(* PLC project TemplatePLC210_03, CODESYS CODESYS V3.5 SP14 Patch 3 *)
(* stored: creationDateTime 2022-10-11T10:43:14.2578546, version 3.5.14.30, modificationDateTime 2022-10-11T10:23:43.7157386, organization Production association OWEN *)

TYPE CTRL8 : STRUCT
  ID : BYTE := 108;
  SIZE : BYTE;
  BIT0 : BIT;
  BIT1 : BIT;
  BIT2 : BIT;
  BIT3 : BIT;
  BIT4 : BIT;
  BIT5 : BIT;
  BIT6 : BIT;
  BIT7 : BIT;
  BIT8 : BIT;
  BIT9 : BIT;
  BIT10 : BIT;
  BIT11 : BIT;
  BIT12 : BIT;
  BIT13 : BIT;
  BIT14 : BIT;
  BIT15 : BIT;
END_STRUCT;
END_TYPE

TYPE bCTRL8 : STRUCT
  CTRL : ARRAY[0..3] OF BYTE;
END_STRUCT;
END_TYPE

TYPE CTRL16 : STRUCT
  ID : WORD := 116;
  SIZE : WORD;
  BIT0 : BIT;
  BIT1 : BIT;
  BIT2 : BIT;
  BIT3 : BIT;
  BIT4 : BIT;
  BIT5 : BIT;
  BIT6 : BIT;
  BIT7 : BIT;
  BIT8 : BIT;
  BIT9 : BIT;
  BIT10 : BIT;
  BIT11 : BIT;
  BIT12 : BIT;
  BIT13 : BIT;
  BIT14 : BIT;
  BIT15 : BIT;
  BIT16 : BIT;
  BIT17 : BIT;
  BIT18 : BIT;
  BIT19 : BIT;
  BIT20 : BIT;
  BIT21 : BIT;
  BIT22 : BIT;
  BIT23 : BIT;
  BIT24 : BIT;
  BIT25 : BIT;
  BIT26 : BIT;
  BIT27 : BIT;
  BIT28 : BIT;
  BIT29 : BIT;
  BIT30 : BIT;
  BIT31 : BIT;
END_STRUCT;
END_TYPE

TYPE wCTRL16 : STRUCT
  CTRL : ARRAY[0..3] OF WORD;
END_STRUCT;
END_TYPE

TYPE CTRL32 : STRUCT
  ID : DWORD := 132;
  SIZE : DWORD;
  BIT0 : BIT;
  BIT1 : BIT;
  BIT2 : BIT;
  BIT3 : BIT;
  BIT4 : BIT;
  BIT5 : BIT;
  BIT6 : BIT;
  BIT7 : BIT;
  BIT8 : BIT;
  BIT9 : BIT;
  BIT10 : BIT;
  BIT11 : BIT;
  BIT12 : BIT;
  BIT13 : BIT;
  BIT14 : BIT;
  BIT15 : BIT;
  BIT16 : BIT;
  BIT17 : BIT;
  BIT18 : BIT;
  BIT19 : BIT;
  BIT20 : BIT;
  BIT21 : BIT;
  BIT22 : BIT;
  BIT23 : BIT;
  BIT24 : BIT;
  BIT25 : BIT;
  BIT26 : BIT;
  BIT27 : BIT;
  BIT28 : BIT;
  BIT29 : BIT;
  BIT30 : BIT;
  BIT31 : BIT;
  BIT32 : BIT;
  BIT33 : BIT;
  BIT34 : BIT;
  BIT35 : BIT;
  BIT36 : BIT;
  BIT37 : BIT;
  BIT38 : BIT;
  BIT39 : BIT;
  BIT40 : BIT;
  BIT41 : BIT;
  BIT42 : BIT;
  BIT43 : BIT;
  BIT44 : BIT;
  BIT45 : BIT;
  BIT46 : BIT;
  BIT47 : BIT;
  BIT48 : BIT;
  BIT49 : BIT;
  BIT50 : BIT;
  BIT51 : BIT;
  BIT52 : BIT;
  BIT53 : BIT;
  BIT54 : BIT;
  BIT55 : BIT;
  BIT56 : BIT;
  BIT57 : BIT;
  BIT58 : BIT;
  BIT59 : BIT;
  BIT60 : BIT;
  BIT61 : BIT;
  BIT62 : BIT;
  BIT63 : BIT;
END_STRUCT;
END_TYPE

TYPE dwCTRL32 : STRUCT
  CTRL : ARRAY[0..3] OF DWORD;
END_STRUCT;
END_TYPE

TYPE uCTRL8 : UNION
  _CTRL8 : CTRL8;
  _wCTRL8 : bCTRL8;
END_UNION;
END_TYPE

TYPE uCTRL16 : UNION
  _CTRL16 : CTRL16;
  _wCTRL16 : wCTRL16;
END_UNION;
END_TYPE

TYPE uCTRL32 : UNION
  _CTRL32 : CTRL32;
  _dwCTRL32 : dwCTRL32;
END_UNION;
END_TYPE

FUNCTION AND16 : BOOL
  VAR_INPUT
    IN_ADR1 : POINTER TO WORD;
    IN_ADR2 : POINTER TO WORD;
    OUT_ADR3 : POINTER TO WORD;
  END_VAR
  VAR
    SIZE : WORD;
    pwADR1 : POINTER TO WORD;
    pwADR2 : POINTER TO WORD;
    pwADR3 : POINTER TO WORD;
    COUNT : WORD;
  END_VAR
  VAR CONSTANT
    STEP : WORD := 2;
  END_VAR

            	pwADR1	:=	IN_ADR1+STEP;
	SIZE	:=	pwADR1^;
IF IN_ADR1^ = IN_ADR2^ AND IN_ADR1^ = OUT_ADR3^ AND SIZE MOD STEP = 0 THEN
	FOR COUNT:=2*STEP TO SIZE-STEP BY STEP DO
		pwADR1	:=	IN_ADR1+COUNT;
		pwADR2	:=	IN_ADR2+COUNT;
		pwADR3	:=	OUT_ADR3+COUNT;
		pwADR3^ := pwADR1^ AND pwADR2^;
	END_FOR
ELSE
	AND16	:=	TRUE;
END_IF

          
END_FUNCTION

FUNCTION AND32 : BOOL
  VAR_INPUT
    IN_ADR1 : POINTER TO DWORD;
    IN_ADR2 : POINTER TO DWORD;
    OUT_ADR3 : POINTER TO DWORD;
  END_VAR
  VAR
    SIZE : DWORD;
    pdwADR1 : POINTER TO DWORD;
    pdwADR2 : POINTER TO DWORD;
    pdwADR3 : POINTER TO DWORD;
    COUNT : DWORD;
  END_VAR
  VAR CONSTANT
    STEP : DWORD := 4;
  END_VAR

            	pdwADR1	:=	IN_ADR1+STEP;
	SIZE	:=	pdwADR1^;
IF IN_ADR1^ = IN_ADR2^ AND IN_ADR1^ = OUT_ADR3^ AND SIZE MOD STEP = 0 THEN
	FOR COUNT:=2*STEP TO SIZE-STEP BY STEP DO
		pdwADR1	:=	IN_ADR1+COUNT;
		pdwADR2	:=	IN_ADR2+COUNT;
		pdwADR3	:=	OUT_ADR3+COUNT;
		pdwADR3^ := pdwADR1^ AND pdwADR2^;
	END_FOR
ELSE
	AND32	:=	TRUE;
END_IF
          
END_FUNCTION

FUNCTION AND8 : BOOL
  VAR_INPUT
    IN_ADR1 : POINTER TO BYTE;
    IN_ADR2 : POINTER TO BYTE;
    OUT_ADR3 : POINTER TO BYTE;
  END_VAR
  VAR
    SIZE : BYTE;
    pbADR1 : POINTER TO BYTE;
    pbADR2 : POINTER TO BYTE;
    pbADR3 : POINTER TO BYTE;
    COUNT : BYTE;
  END_VAR

            IF IN_ADR1^ = IN_ADR2^ AND IN_ADR1^ = OUT_ADR3^ THEN
	pbADR1	:=	IN_ADR1+1;
	SIZE	:=	pbADR1^;
	FOR COUNT:=2 TO SIZE-1 DO
		pbADR1	:=	IN_ADR1+COUNT;
		pbADR2	:=	IN_ADR2+COUNT;
		pbADR3	:=	OUT_ADR3+COUNT;
		pbADR3^ := pbADR1^ AND pbADR2^;
	END_FOR
ELSE
	AND8	:=	TRUE;
END_IF

          
END_FUNCTION

FUNCTION NAND8 : BOOL
  VAR_INPUT
    IN_ADR1 : POINTER TO BYTE;
    IN_ADR2 : POINTER TO BYTE;
    OUT_ADR3 : POINTER TO BYTE;
  END_VAR
  VAR
    SIZE : BYTE;
    pbADR1 : POINTER TO BYTE;
    pbADR2 : POINTER TO BYTE;
    pbADR3 : POINTER TO BYTE;
    COUNT : BYTE;
  END_VAR

            IF IN_ADR1^ = IN_ADR2^ AND IN_ADR1^ = OUT_ADR3^ THEN
	pbADR1	:=	IN_ADR1+1;
	SIZE	:=	pbADR1^;
	FOR COUNT:=2 TO SIZE-1 DO
		pbADR1	:=	IN_ADR1+COUNT;
		pbADR2	:=	IN_ADR2+COUNT;
		pbADR3	:=	OUT_ADR3+COUNT;
		pbADR3^ := NOT(pbADR1^ AND pbADR2^);
	END_FOR
ELSE
	NAND8	:=	TRUE;
END_IF

          
END_FUNCTION

FUNCTION NAND16 : BOOL
  VAR_INPUT
    IN_ADR1 : POINTER TO WORD;
    IN_ADR2 : POINTER TO WORD;
    OUT_ADR3 : POINTER TO WORD;
  END_VAR
  VAR
    SIZE : WORD;
    pwADR1 : POINTER TO WORD;
    pwADR2 : POINTER TO WORD;
    pwADR3 : POINTER TO WORD;
    COUNT : WORD;
  END_VAR
  VAR CONSTANT
    STEP : WORD := 2;
  END_VAR

            	pwADR1	:=	IN_ADR1+STEP;
	SIZE	:=	pwADR1^;
IF IN_ADR1^ = IN_ADR2^ AND IN_ADR1^ = OUT_ADR3^ AND SIZE MOD STEP = 0 THEN
	FOR COUNT:=2*STEP TO SIZE-STEP BY STEP DO
		pwADR1	:=	IN_ADR1+COUNT;
		pwADR2	:=	IN_ADR2+COUNT;
		pwADR3	:=	OUT_ADR3+COUNT;
		pwADR3^ := NOT(pwADR1^ AND pwADR2^);
	END_FOR
ELSE
	NAND16	:=	TRUE;
END_IF

          
END_FUNCTION

FUNCTION NAND32 : BOOL
  VAR_INPUT
    IN_ADR1 : POINTER TO DWORD;
    IN_ADR2 : POINTER TO DWORD;
    OUT_ADR3 : POINTER TO DWORD;
  END_VAR
  VAR
    SIZE : DWORD;
    pdwADR1 : POINTER TO DWORD;
    pdwADR2 : POINTER TO DWORD;
    pdwADR3 : POINTER TO DWORD;
    COUNT : DWORD;
  END_VAR
  VAR CONSTANT
    STEP : DWORD := 4;
  END_VAR

            	pdwADR1	:=	IN_ADR1+STEP;
	SIZE	:=	pdwADR1^;
IF IN_ADR1^ = IN_ADR2^ AND IN_ADR1^ = OUT_ADR3^ AND SIZE MOD STEP = 0 THEN
	FOR COUNT:=2*STEP TO SIZE-STEP BY STEP DO
		pdwADR1	:=	IN_ADR1+COUNT;
		pdwADR2	:=	IN_ADR2+COUNT;
		pdwADR3	:=	OUT_ADR3+COUNT;
		pdwADR3^ := NOT(pdwADR1^ AND pdwADR2^);
	END_FOR
ELSE
	NAND32	:=	TRUE;
END_IF

          
END_FUNCTION

FUNCTION OR8 : BOOL
  VAR_INPUT
    IN_ADR1 : POINTER TO BYTE;
    IN_ADR2 : POINTER TO BYTE;
    OUT_ADR3 : POINTER TO BYTE;
  END_VAR
  VAR
    SIZE : BYTE;
    pbADR1 : POINTER TO BYTE;
    pbADR2 : POINTER TO BYTE;
    pbADR3 : POINTER TO BYTE;
    COUNT : BYTE;
  END_VAR

            IF IN_ADR1^ = IN_ADR2^ AND IN_ADR1^ = OUT_ADR3^ THEN
	pbADR1	:=	IN_ADR1+1;
	SIZE	:=	pbADR1^;
	FOR COUNT:=2 TO SIZE-1 DO
		pbADR1	:=	IN_ADR1+COUNT;
		pbADR2	:=	IN_ADR2+COUNT;
		pbADR3	:=	OUT_ADR3+COUNT;
		pbADR3^ := pbADR1^ OR pbADR2^;
	END_FOR
ELSE
	OR8	:=	TRUE;
END_IF

          
END_FUNCTION

FUNCTION OR16 : BOOL
  VAR_INPUT
    IN_ADR1 : POINTER TO WORD;
    IN_ADR2 : POINTER TO WORD;
    OUT_ADR3 : POINTER TO WORD;
  END_VAR
  VAR
    SIZE : WORD;
    pwADR1 : POINTER TO WORD;
    pwADR2 : POINTER TO WORD;
    pwADR3 : POINTER TO WORD;
    COUNT : WORD;
  END_VAR
  VAR CONSTANT
    STEP : WORD := 2;
  END_VAR

            	pwADR1	:=	IN_ADR1+STEP;
	SIZE	:=	pwADR1^;
IF IN_ADR1^ = IN_ADR2^ AND IN_ADR1^ = OUT_ADR3^ AND SIZE MOD STEP = 0 THEN
	FOR COUNT:=2*STEP TO SIZE-STEP BY STEP DO
		pwADR1	:=	IN_ADR1+COUNT;
		pwADR2	:=	IN_ADR2+COUNT;
		pwADR3	:=	OUT_ADR3+COUNT;
		pwADR3^ := pwADR1^ OR pwADR2^;
	END_FOR
ELSE
	OR16	:=	TRUE;
END_IF

          
END_FUNCTION

FUNCTION OR32 : BOOL
  VAR_INPUT
    IN_ADR1 : POINTER TO DWORD;
    IN_ADR2 : POINTER TO DWORD;
    OUT_ADR3 : POINTER TO DWORD;
  END_VAR
  VAR
    SIZE : DWORD;
    pdwADR1 : POINTER TO DWORD;
    pdwADR2 : POINTER TO DWORD;
    pdwADR3 : POINTER TO DWORD;
    COUNT : DWORD;
  END_VAR
  VAR CONSTANT
    STEP : DWORD := 4;
  END_VAR

            	pdwADR1	:=	IN_ADR1+STEP;
	SIZE	:=	pdwADR1^;
IF IN_ADR1^ = IN_ADR2^ AND IN_ADR1^ = OUT_ADR3^ AND SIZE MOD STEP = 0 THEN
	FOR COUNT:=2*STEP TO SIZE-STEP BY STEP DO
		pdwADR1	:=	IN_ADR1+COUNT;
		pdwADR2	:=	IN_ADR2+COUNT;
		pdwADR3	:=	OUT_ADR3+COUNT;
		pdwADR3^ := pdwADR1^ OR pdwADR2^;
	END_FOR
ELSE
	OR32	:=	TRUE;
END_IF

          
END_FUNCTION

FUNCTION NOR8 : BOOL
  VAR_INPUT
    IN_ADR1 : POINTER TO BYTE;
    IN_ADR2 : POINTER TO BYTE;
    OUT_ADR3 : POINTER TO BYTE;
  END_VAR
  VAR
    SIZE : BYTE;
    pbADR1 : POINTER TO BYTE;
    pbADR2 : POINTER TO BYTE;
    pbADR3 : POINTER TO BYTE;
    COUNT : BYTE;
  END_VAR

            IF IN_ADR1^ = IN_ADR2^ AND IN_ADR1^ = OUT_ADR3^ THEN
	pbADR1	:=	IN_ADR1+1;
	SIZE	:=	pbADR1^;
	FOR COUNT:=2 TO SIZE-1 DO
		pbADR1	:=	IN_ADR1+COUNT;
		pbADR2	:=	IN_ADR2+COUNT;
		pbADR3	:=	OUT_ADR3+COUNT;
		pbADR3^ := NOT(pbADR1^ OR pbADR2^);
	END_FOR
ELSE
	NOR8	:=	TRUE;
END_IF

          
END_FUNCTION

FUNCTION NOR16 : BOOL
  VAR_INPUT
    IN_ADR1 : POINTER TO WORD;
    IN_ADR2 : POINTER TO WORD;
    OUT_ADR3 : POINTER TO WORD;
  END_VAR
  VAR
    SIZE : WORD;
    pwADR1 : POINTER TO WORD;
    pwADR2 : POINTER TO WORD;
    pwADR3 : POINTER TO WORD;
    COUNT : WORD;
  END_VAR
  VAR CONSTANT
    STEP : WORD := 2;
  END_VAR

            	pwADR1	:=	IN_ADR1+STEP;
	SIZE	:=	pwADR1^;
IF IN_ADR1^ = IN_ADR2^ AND IN_ADR1^ = OUT_ADR3^ AND SIZE MOD STEP = 0 THEN
	FOR COUNT:=2*STEP TO SIZE-STEP BY STEP DO
		pwADR1	:=	IN_ADR1+COUNT;
		pwADR2	:=	IN_ADR2+COUNT;
		pwADR3	:=	OUT_ADR3+COUNT;
		pwADR3^ := NOT(pwADR1^ OR pwADR2^);
	END_FOR
ELSE
	NOR16	:=	TRUE;
END_IF

          
END_FUNCTION

FUNCTION NOR32 : BOOL
  VAR_INPUT
    IN_ADR1 : POINTER TO DWORD;
    IN_ADR2 : POINTER TO DWORD;
    OUT_ADR3 : POINTER TO DWORD;
  END_VAR
  VAR
    SIZE : DWORD;
    pdwADR1 : POINTER TO DWORD;
    pdwADR2 : POINTER TO DWORD;
    pdwADR3 : POINTER TO DWORD;
    COUNT : DWORD;
  END_VAR
  VAR CONSTANT
    STEP : DWORD := 4;
  END_VAR

            	pdwADR1	:=	IN_ADR1+STEP;
	SIZE	:=	pdwADR1^;
IF IN_ADR1^ = IN_ADR2^ AND IN_ADR1^ = OUT_ADR3^ AND SIZE MOD STEP = 0 THEN
	FOR COUNT:=2*STEP TO SIZE-STEP BY STEP DO
		pdwADR1	:=	IN_ADR1+COUNT;
		pdwADR2	:=	IN_ADR2+COUNT;
		pdwADR3	:=	OUT_ADR3+COUNT;
		pdwADR3^ := NOT(pdwADR1^ OR pdwADR2^);
	END_FOR
ELSE
	NOR32	:=	TRUE;
END_IF

          
END_FUNCTION

FUNCTION XOR8 : BOOL
  VAR_INPUT
    IN_ADR1 : POINTER TO BYTE;
    IN_ADR2 : POINTER TO BYTE;
    OUT_ADR3 : POINTER TO BYTE;
  END_VAR
  VAR
    SIZE : BYTE;
    pbADR1 : POINTER TO BYTE;
    pbADR2 : POINTER TO BYTE;
    pbADR3 : POINTER TO BYTE;
    COUNT : BYTE;
  END_VAR

            IF IN_ADR1^ = IN_ADR2^ AND IN_ADR1^ = OUT_ADR3^ THEN
	pbADR1	:=	IN_ADR1+1;
	SIZE	:=	pbADR1^;
	FOR COUNT:=2 TO SIZE-1 DO
		pbADR1	:=	IN_ADR1+COUNT;
		pbADR2	:=	IN_ADR2+COUNT;
		pbADR3	:=	OUT_ADR3+COUNT;
		pbADR3^ := pbADR1^ XOR pbADR2^;
	END_FOR
ELSE
	XOR8	:=	TRUE;
END_IF

          
END_FUNCTION

FUNCTION XOR16 : BOOL
  VAR_INPUT
    IN_ADR1 : POINTER TO WORD;
    IN_ADR2 : POINTER TO WORD;
    OUT_ADR3 : POINTER TO WORD;
  END_VAR
  VAR
    SIZE : WORD;
    pwADR1 : POINTER TO WORD;
    pwADR2 : POINTER TO WORD;
    pwADR3 : POINTER TO WORD;
    COUNT : WORD;
  END_VAR
  VAR CONSTANT
    STEP : WORD := 2;
  END_VAR

            	pwADR1	:=	IN_ADR1+STEP;
	SIZE	:=	pwADR1^;
IF IN_ADR1^ = IN_ADR2^ AND IN_ADR1^ = OUT_ADR3^ AND SIZE MOD STEP = 0 THEN
	FOR COUNT:=2*STEP TO SIZE-STEP BY STEP DO
		pwADR1	:=	IN_ADR1+COUNT;
		pwADR2	:=	IN_ADR2+COUNT;
		pwADR3	:=	OUT_ADR3+COUNT;
		pwADR3^ := pwADR1^ XOR pwADR2^;
	END_FOR
ELSE
	XOR16	:=	TRUE;
END_IF

          
END_FUNCTION

FUNCTION XOR32 : BOOL
  VAR_INPUT
    IN_ADR1 : POINTER TO DWORD;
    IN_ADR2 : POINTER TO DWORD;
    OUT_ADR3 : POINTER TO DWORD;
  END_VAR
  VAR
    SIZE : DWORD;
    pdwADR1 : POINTER TO DWORD;
    pdwADR2 : POINTER TO DWORD;
    pdwADR3 : POINTER TO DWORD;
    COUNT : DWORD;
  END_VAR
  VAR CONSTANT
    STEP : DWORD := 4;
  END_VAR

            	pdwADR1	:=	IN_ADR1+STEP;
	SIZE	:=	pdwADR1^;
IF IN_ADR1^ = IN_ADR2^ AND IN_ADR1^ = OUT_ADR3^ AND SIZE MOD STEP = 0 THEN
	FOR COUNT:=2*STEP TO SIZE-STEP BY STEP DO
		pdwADR1	:=	IN_ADR1+COUNT;
		pdwADR2	:=	IN_ADR2+COUNT;
		pdwADR3	:=	OUT_ADR3+COUNT;
		pdwADR3^ := pdwADR1^ XOR pdwADR2^;
	END_FOR
ELSE
	XOR32	:=	TRUE;
END_IF

          
END_FUNCTION

FUNCTION NXOR8 : BOOL
  VAR_INPUT
    IN_ADR1 : POINTER TO BYTE;
    IN_ADR2 : POINTER TO BYTE;
    OUT_ADR3 : POINTER TO BYTE;
  END_VAR
  VAR
    SIZE : BYTE;
    pbADR1 : POINTER TO BYTE;
    pbADR2 : POINTER TO BYTE;
    pbADR3 : POINTER TO BYTE;
    COUNT : BYTE;
  END_VAR

            IF IN_ADR1^ = IN_ADR2^ AND IN_ADR1^ = OUT_ADR3^ THEN
	pbADR1	:=	IN_ADR1+1;
	SIZE	:=	pbADR1^;
	FOR COUNT:=2 TO SIZE-1 DO
		pbADR1	:=	IN_ADR1+COUNT;
		pbADR2	:=	IN_ADR2+COUNT;
		pbADR3	:=	OUT_ADR3+COUNT;
		pbADR3^ := NOT(pbADR1^ XOR pbADR2^);
	END_FOR
ELSE
	NXOR8	:=	TRUE;
END_IF

          
END_FUNCTION

FUNCTION NXOR16 : BOOL
  VAR_INPUT
    IN_ADR1 : POINTER TO WORD;
    IN_ADR2 : POINTER TO WORD;
    OUT_ADR3 : POINTER TO WORD;
  END_VAR
  VAR
    SIZE : WORD;
    pwADR1 : POINTER TO WORD;
    pwADR2 : POINTER TO WORD;
    pwADR3 : POINTER TO WORD;
    COUNT : WORD;
  END_VAR
  VAR CONSTANT
    STEP : WORD := 2;
  END_VAR

            	pwADR1	:=	IN_ADR1+STEP;
	SIZE	:=	pwADR1^;
IF IN_ADR1^ = IN_ADR2^ AND IN_ADR1^ = OUT_ADR3^ AND SIZE MOD STEP = 0 THEN
	FOR COUNT:=2*STEP TO SIZE-STEP BY STEP DO
		pwADR1	:=	IN_ADR1+COUNT;
		pwADR2	:=	IN_ADR2+COUNT;
		pwADR3	:=	OUT_ADR3+COUNT;
		pwADR3^ := NOT(pwADR1^ XOR pwADR2^);
	END_FOR
ELSE
	NXOR16	:=	TRUE;
END_IF

          
END_FUNCTION

FUNCTION NXOR32 : BOOL
  VAR_INPUT
    IN_ADR1 : POINTER TO DWORD;
    IN_ADR2 : POINTER TO DWORD;
    OUT_ADR3 : POINTER TO DWORD;
  END_VAR
  VAR
    SIZE : DWORD;
    pdwADR1 : POINTER TO DWORD;
    pdwADR2 : POINTER TO DWORD;
    pdwADR3 : POINTER TO DWORD;
    COUNT : DWORD;
  END_VAR
  VAR CONSTANT
    STEP : DWORD := 4;
  END_VAR

            	pdwADR1	:=	IN_ADR1+STEP;
	SIZE	:=	pdwADR1^;
IF IN_ADR1^ = IN_ADR2^ AND IN_ADR1^ = OUT_ADR3^ AND SIZE MOD STEP = 0 THEN
	FOR COUNT:=2*STEP TO SIZE-STEP BY STEP DO
		pdwADR1	:=	IN_ADR1+COUNT;
		pdwADR2	:=	IN_ADR2+COUNT;
		pdwADR3	:=	OUT_ADR3+COUNT;
		pdwADR3^ := NOT(pdwADR1^ XOR pdwADR2^);
	END_FOR
ELSE
	NXOR32	:=	TRUE;
END_IF

          
END_FUNCTION

FUNCTION NOT8 : BOOL
  VAR_INPUT
    IN_ADR1 : POINTER TO BYTE;
    OUT_ADR2 : POINTER TO BYTE;
  END_VAR
  VAR
    SIZE : BYTE;
    pbADR1 : POINTER TO BYTE;
    pbADR2 : POINTER TO BYTE;
    COUNT : BYTE;
  END_VAR

            IF IN_ADR1^ = OUT_ADR2^ THEN
	pbADR1	:=	IN_ADR1+1;
	SIZE	:=	pbADR1^;
	FOR COUNT:=2 TO SIZE-1 DO
		pbADR1	:=	IN_ADR1+COUNT;
		pbADR2	:=	OUT_ADR2+COUNT;
		pbADR2^ := NOT pbADR1^;
	END_FOR
ELSE
	NOT8	:=	TRUE;
END_IF

          
END_FUNCTION

FUNCTION NOT16 : BOOL
  VAR_INPUT
    IN_ADR1 : POINTER TO WORD;
    OUT_ADR2 : POINTER TO WORD;
  END_VAR
  VAR
    SIZE : WORD;
    pwADR1 : POINTER TO WORD;
    pwADR2 : POINTER TO WORD;
    COUNT : WORD;
  END_VAR
  VAR CONSTANT
    STEP : WORD := 2;
  END_VAR

            	pwADR1	:=	IN_ADR1+STEP;
	SIZE	:=	pwADR1^;
IF IN_ADR1^ = OUT_ADR2^ AND SIZE MOD STEP = 0 THEN
	FOR COUNT:=2*STEP TO SIZE-STEP BY STEP DO
		pwADR1	:=	IN_ADR1+COUNT;
		pwADR2	:=	OUT_ADR2+COUNT;
		pwADR2^ := NOT pwADR1^;
	END_FOR
ELSE
	NOT16	:=	TRUE;
END_IF

          
END_FUNCTION

FUNCTION NOT32 : BOOL
  VAR_INPUT
    IN_ADR1 : POINTER TO DWORD;
    OUT_ADR2 : POINTER TO DWORD;
  END_VAR
  VAR
    SIZE : DWORD;
    pdwADR1 : POINTER TO DWORD;
    pdwADR2 : POINTER TO DWORD;
    COUNT : DWORD;
  END_VAR
  VAR CONSTANT
    STEP : DWORD := 4;
  END_VAR

            	pdwADR1	:=	IN_ADR1+STEP;
	SIZE	:=	pdwADR1^;
IF IN_ADR1^ = OUT_ADR2^ AND SIZE MOD STEP = 0 THEN
	FOR COUNT:=2*STEP TO SIZE-STEP BY STEP DO
		pdwADR1	:=	IN_ADR1+COUNT;
		pdwADR2	:=	OUT_ADR2+COUNT;
		pdwADR2^ := NOT pdwADR1^;
	END_FOR
ELSE
	NOT32	:=	TRUE;
END_IF

          
END_FUNCTION

FUNCTION EQ8 : BOOL
  VAR_INPUT
    IN_ADR1 : POINTER TO BYTE;
    IN_ADR2 : POINTER TO BYTE;
    OUT_ADR3 : POINTER TO BYTE;
  END_VAR

            EQ8 := NXOR8(IN_ADR1,IN_ADR2,OUT_ADR3);
          
END_FUNCTION

FUNCTION EQ16 : BOOL
  VAR_INPUT
    IN_ADR1 : POINTER TO BYTE;
    IN_ADR2 : POINTER TO BYTE;
    OUT_ADR3 : POINTER TO BYTE;
  END_VAR

            EQ16 := NXOR16(IN_ADR1,IN_ADR2,OUT_ADR3);
          
END_FUNCTION

FUNCTION EQ32 : BOOL
  VAR_INPUT
    IN_ADR1 : POINTER TO BYTE;
    IN_ADR2 : POINTER TO BYTE;
    OUT_ADR3 : POINTER TO BYTE;
  END_VAR

            EQ32 := NXOR32(IN_ADR1,IN_ADR2,OUT_ADR3);
          
END_FUNCTION

FUNCTION NEQ8 : BOOL
  VAR_INPUT
    IN_ADR1 : POINTER TO BYTE;
    IN_ADR2 : POINTER TO BYTE;
    OUT_ADR3 : POINTER TO BYTE;
  END_VAR

            NEQ8 := XOR8(IN_ADR1,IN_ADR2,OUT_ADR3);
          
END_FUNCTION

FUNCTION NEQ16 : BOOL
  VAR_INPUT
    IN_ADR1 : POINTER TO BYTE;
    IN_ADR2 : POINTER TO BYTE;
    OUT_ADR3 : POINTER TO BYTE;
  END_VAR

            NEQ16 := XOR16(IN_ADR1,IN_ADR2,OUT_ADR3);
          
END_FUNCTION

FUNCTION NEQ32 : BOOL
  VAR_INPUT
    IN_ADR1 : POINTER TO BYTE;
    IN_ADR2 : POINTER TO BYTE;
    OUT_ADR3 : POINTER TO BYTE;
  END_VAR

            NEQ32 := XOR32(IN_ADR1,IN_ADR2,OUT_ADR3);
          
END_FUNCTION

FUNCTION GET_BIT8 : BOOL
  VAR_INPUT
    IN_ADR : POINTER TO BYTE;
    BIT_NUMBER : LINT;
  END_VAR
  VAR
    SIZE : BYTE;
    pbADR : POINTER TO BYTE;
  END_VAR
  VAR CONSTANT
    STEP : BYTE := 1;
  END_VAR

            pbADR	:=	IN_ADR+STEP;
SIZE	:=	pbADR^;
IF BIT_NUMBER >= (SIZE-2*STEP)*8 OR BIT_NUMBER <0 THEN
	BIT_NUMBER	:=	0;
	BIT_NUMBER	:=	BIT_NUMBER/BIT_NUMBER;
	//Ты вышел за пределы структуры, дядь
END_IF
pbADR := IN_ADR + (2 + ANY_TO_DWORD(BIT_NUMBER/8))*STEP;
GET_BIT8 := ANY_TO_BOOL(SHL(1,BIT_NUMBER MOD 8) AND pbADR^);

          
END_FUNCTION

FUNCTION SET_BIT8 : BOOL
  VAR_INPUT
    IN_ADR : POINTER TO BYTE;
    BIT_NUMBER : LINT;
  END_VAR
  VAR
    SIZE : BYTE;
    pbADR : POINTER TO BYTE;
    bBYTE : BYTE;
  END_VAR
  VAR CONSTANT
    STEP : BYTE := 1;
    STEP_SIZE : BYTE := (STEP * 8);
  END_VAR

            pbADR:=	IN_ADR+STEP;
SIZE	:=	pbADR^;	
IF BIT_NUMBER >= (SIZE-2*STEP)*8 OR BIT_NUMBER <0 THEN
	BIT_NUMBER	:=	0;
	BIT_NUMBER	:=	BIT_NUMBER/BIT_NUMBER;
	//Ты вышел за пределы структуры, дядь
END_IF
pbADR := IN_ADR + 2*STEP + ANY_TO_DWORD(BIT_NUMBER/STEP_SIZE);
bBYTE:=SHL(1,BIT_NUMBER MOD STEP_SIZE);
pbADR^ := pbADR^ OR bBYTE;
          
END_FUNCTION

FUNCTION FIND1ST_0_8 : LINT
  VAR_INPUT
    IN_ADR1 : POINTER TO BYTE;
  END_VAR
  VAR
    SIZE : BYTE;
    pbADR1 : POINTER TO BYTE;
    COUNT : BYTE;
  END_VAR
  VAR CONSTANT
    ONE : BYTE := 1;
  END_VAR

            pbADR1	:=	IN_ADR1+1;
SIZE	:=	pbADR1^;
FOR COUNT:=2 TO SIZE-1 DO
	pbADR1	:=	IN_ADR1+COUNT;
	IF pbADR1^ =0 THEN
		RETURN;
	ELSE
		REPEAT
 			IF	NOT((NOT(SHL(ONE,FIND1ST_0_8 MOD 8)) OR pbADR1^ )= 255) THEN			
				RETURN; 		
			END_IF;
			FIND1ST_0_8:=FIND1ST_0_8 + 1;
		UNTIL FIND1ST_0_8 MOD 8 = 0
		END_REPEAT;	
	END_IF
END_FOR
FIND1ST_0_8:=-1;
          
END_FUNCTION

FUNCTION FIND1ST_1_8 : LINT
  VAR_INPUT
    IN_ADR1 : POINTER TO BYTE;
  END_VAR
  VAR
    SIZE : BYTE;
    pbADR1 : POINTER TO BYTE;
    COUNT : BYTE;
  END_VAR
  VAR CONSTANT
    ONE : BYTE := 1;
    STEP : BYTE := 1;
    STEP_SIZE : BYTE := (STEP * 8);
  END_VAR

            pbADR1	:=	IN_ADR1+STEP;
SIZE	:=	pbADR1^;
FOR COUNT:=2 TO SIZE-1 DO
	pbADR1	:=	IN_ADR1+COUNT;
	IF NOT(pbADR1^ =0) THEN
		REPEAT
 			IF	(NOT(SHL(ONE,FIND1ST_1_8 MOD 8)) OR pbADR1^ )= 255 THEN
				RETURN;
			END_IF;
			FIND1ST_1_8:=FIND1ST_1_8 + 1;
		UNTIL FIND1ST_1_8 MOD 8 = 0
		END_REPEAT;
	ELSE
		FIND1ST_1_8:=FIND1ST_1_8 + 8;
	END_IF
END_FOR
FIND1ST_1_8:=-1;
          
END_FUNCTION

FUNCTION GET_BIT16 : BOOL
  VAR_INPUT
    IN_ADR : POINTER TO WORD;
    BIT_NUMBER : LINT;
  END_VAR
  VAR
    SIZE : WORD;
    pwADR : POINTER TO WORD;
  END_VAR
  VAR CONSTANT
    STEP : WORD := 2;
    STEP_SIZE : WORD := (STEP * 8);
  END_VAR

            pwADR	:=	IN_ADR+STEP;
SIZE	:=	pwADR^;
IF BIT_NUMBER >= (SIZE-2*STEP)*8 OR BIT_NUMBER <0 THEN
	BIT_NUMBER	:=	0;
	BIT_NUMBER	:=	BIT_NUMBER/BIT_NUMBER;
	//Ты вышел за пределы структуры, дядь
END_IF
pwADR := IN_ADR + (2 + ANY_TO_DWORD(BIT_NUMBER/STEP_SIZE))*STEP;
GET_BIT16 := ANY_TO_BOOL(SHL(1,BIT_NUMBER MOD STEP_SIZE) AND pwADR^);

          
END_FUNCTION

FUNCTION GET_BIT32 : BOOL
  VAR_INPUT
    IN_ADR : POINTER TO DWORD;
    BIT_NUMBER : LINT;
  END_VAR
  VAR
    SIZE : DWORD;
    pdwADR : POINTER TO DWORD;
  END_VAR
  VAR CONSTANT
    STEP : DWORD := 4;
    STEP_SIZE : DWORD := (STEP * 8);
  END_VAR

            pdwADR	:=	IN_ADR+STEP;
SIZE	:=	pdwADR^;
IF BIT_NUMBER >= (SIZE-2*STEP)*8 OR BIT_NUMBER <0 THEN
	BIT_NUMBER	:=	0;
	BIT_NUMBER	:=	BIT_NUMBER/BIT_NUMBER;
	//Ты вышел за пределы структуры, дядь
END_IF
pdwADR := IN_ADR + (2 + ANY_TO_DWORD(BIT_NUMBER/STEP_SIZE))*STEP;
GET_BIT32 := ANY_TO_BOOL(SHL(1,BIT_NUMBER MOD STEP_SIZE) AND pdwADR^);

          
END_FUNCTION

FUNCTION SET_BIT16 : BOOL
  VAR_INPUT
    IN_ADR : POINTER TO WORD;
    BIT_NUMBER : LINT;
  END_VAR
  VAR
    SIZE : WORD;
    pwADR : POINTER TO WORD;
    wWORD : WORD;
  END_VAR
  VAR CONSTANT
    STEP : WORD := 2;
    STEP_SIZE : WORD := (STEP * 8);
  END_VAR

            pwADR:=	IN_ADR+STEP;
SIZE	:=	pwADR^;	
IF BIT_NUMBER >= (SIZE-2*STEP)*8 OR BIT_NUMBER <0 THEN
	BIT_NUMBER	:=	0;
	BIT_NUMBER	:=	BIT_NUMBER/BIT_NUMBER;
	//Ты вышел за пределы структуры, дядь
END_IF
pwADR := IN_ADR + (2 + ANY_TO_DWORD(BIT_NUMBER/STEP_SIZE))*STEP;
wWORD:=SHL(1,BIT_NUMBER MOD STEP_SIZE);
pwADR^ := pwADR^ OR wWORD;
          
END_FUNCTION

FUNCTION SET_BIT32 : BOOL
  VAR_INPUT
    IN_ADR : POINTER TO DWORD;
    BIT_NUMBER : LINT;
  END_VAR
  VAR
    SIZE : DWORD;
    pdwADR : POINTER TO DWORD;
    dwDWORD : DWORD;
  END_VAR
  VAR CONSTANT
    STEP : WORD := 4;
    STEP_SIZE : WORD := (STEP * 8);
  END_VAR

            pdwADR:=	IN_ADR+STEP;
SIZE	:=	pdwADR^;	
IF BIT_NUMBER >= (SIZE-2*STEP)*8 OR BIT_NUMBER <0 THEN
	BIT_NUMBER	:=	0;
	BIT_NUMBER	:=	BIT_NUMBER/BIT_NUMBER;
	//Ты вышел за пределы структуры, дядь
END_IF
pdwADR := IN_ADR + (2 + ANY_TO_DWORD(BIT_NUMBER/STEP_SIZE))*STEP;
dwDWORD:=SHL(1,BIT_NUMBER MOD STEP_SIZE);
pdwADR^ := pdwADR^ OR dwDWORD;	
          
END_FUNCTION

PROGRAM CHECK_FIND1ST_1_16
  VAR
    CTRL1 : uCTRL16;
    N : LINT;
  END_VAR

            CTRL1._CTRL16.SIZE:=ANY_TO_WORD(SIZEOF(CTRL1));
N:=FIND1ST_1_16(ADR(CTRL1));
          
END_PROGRAM

FUNCTION FIND1ST_0_16 : LINT
  VAR_INPUT
    IN_ADR1 : POINTER TO WORD;
  END_VAR
  VAR
    SIZE : WORD;
    pwADR1 : POINTER TO WORD;
    COUNT : WORD;
  END_VAR
  VAR CONSTANT
    ONE : WORD := 1;
    STEP : WORD := 2;
    STEP_SIZE : WORD := (STEP * 8);
  END_VAR

            pwADR1	:=	IN_ADR1+STEP;
SIZE	:=	pwADR1^;
FOR COUNT:=2*STEP TO SIZE-1 BY STEP DO
	pwADR1	:=	IN_ADR1+COUNT;
	IF pwADR1^ =0 THEN
		RETURN;
	ELSE
		REPEAT
 			IF	NOT((NOT(SHL(ONE,FIND1ST_0_16 MOD STEP_SIZE)) OR pwADR1^ )= 65535) THEN		
				RETURN; 		
			END_IF;
			FIND1ST_0_16:=FIND1ST_0_16 + 1;
		UNTIL FIND1ST_0_16 MOD STEP_SIZE = 0
		END_REPEAT;	
	END_IF
END_FOR
FIND1ST_0_16:=-1;
          
END_FUNCTION

FUNCTION FIND1ST_0_32 : LINT
  VAR_INPUT
    IN_ADR1 : POINTER TO DWORD;
  END_VAR
  VAR
    SIZE : DWORD;
    pdwADR1 : POINTER TO DWORD;
    COUNT : DWORD;
  END_VAR
  VAR CONSTANT
    ONE : DWORD := 1;
    STEP : DWORD := 4;
    STEP_SIZE : DWORD := (STEP * 8);
  END_VAR

            pdwADR1	:=	IN_ADR1+STEP;
SIZE	:=	pdwADR1^;
FOR COUNT:=2*STEP TO SIZE-1 BY STEP DO
	pdwADR1	:=	IN_ADR1+COUNT;
	IF pdwADR1^ =0 THEN
		RETURN;
	ELSE
		REPEAT
 			IF	NOT((NOT(SHL(ONE,FIND1ST_0_32 MOD STEP_SIZE)) OR pdwADR1^ )= 4294967295) THEN		
				RETURN; 		
			END_IF;
			FIND1ST_0_32:=FIND1ST_0_32 + 1;
		UNTIL FIND1ST_0_32 MOD STEP_SIZE = 0
		END_REPEAT;	
	END_IF
END_FOR
FIND1ST_0_32:=-1;
          
END_FUNCTION

FUNCTION FIND1ST_1_16 : LINT
  VAR_INPUT
    IN_ADR1 : POINTER TO WORD;
  END_VAR
  VAR
    SIZE : WORD;
    pwADR1 : POINTER TO WORD;
    COUNT : WORD;
  END_VAR
  VAR CONSTANT
    ONE : WORD := 1;
    STEP : WORD := 2;
    STEP_SIZE : WORD := (STEP * 8);
  END_VAR

            pwADR1	:=	IN_ADR1+STEP;
SIZE	:=	pwADR1^;
FOR COUNT:=2*STEP TO SIZE-STEP BY STEP DO
	pwADR1	:=	IN_ADR1+COUNT;
	IF NOT(pwADR1^ =0) THEN
		REPEAT
 			IF	(NOT(SHL(ONE,FIND1ST_1_16 MOD STEP_SIZE)) OR pwADR1^ )= 65535 THEN
				RETURN;
			END_IF;
			FIND1ST_1_16:=FIND1ST_1_16 + 1;
		UNTIL FIND1ST_1_16 MOD STEP_SIZE = 0
		END_REPEAT;
	ELSE
		FIND1ST_1_16:=FIND1ST_1_16 + STEP_SIZE;
	END_IF
END_FOR
FIND1ST_1_16:=-1;
          
END_FUNCTION

FUNCTION FIND1ST_1_32 : LINT
  VAR_INPUT
    IN_ADR1 : POINTER TO WORD;
  END_VAR
  VAR
    SIZE : DWORD;
    pdwADR1 : POINTER TO DWORD;
    COUNT : DWORD;
  END_VAR
  VAR CONSTANT
    ONE : DWORD := 1;
    STEP : DWORD := 4;
    STEP_SIZE : DWORD := (STEP * 8);
  END_VAR

            pdwADR1	:=	IN_ADR1+STEP;
SIZE	:=	pdwADR1^;
FOR COUNT:=2*STEP TO SIZE-1 BY STEP DO
	pdwADR1	:=	IN_ADR1+COUNT;
	IF NOT(pdwADR1^ =0) THEN
		REPEAT
 			IF	(NOT(SHL(ONE,FIND1ST_1_32 MOD STEP_SIZE)) OR pdwADR1^ )= 4294967295 THEN
				RETURN;
			END_IF;
			FIND1ST_1_32:=FIND1ST_1_32 + 1;
		UNTIL FIND1ST_1_32 MOD STEP_SIZE = 0
		END_REPEAT;
	ELSE
		FIND1ST_1_32:=FIND1ST_1_32 + STEP_SIZE;
	END_IF
END_FOR
FIND1ST_1_32:=-1;
          
END_FUNCTION

PROGRAM CHECK_AND8
  VAR
    CTRL1 : uCTRL8;
    CTRL2 : uCTRL8;
    CTRL3 : uCTRL8;
    TIMER : TON;
    STAGE : ENUM;
    N : LINT;
    X1 : BOOL;
    X2 : BOOL;
    X3 : BOOL;
    CORRECT : BOOL := TRUE;
  END_VAR

            CTRL1._CTRL8.SIZE:=ANY_TO_BYTE(SIZEOF(CTRL1));
CTRL2._CTRL8.SIZE:=ANY_TO_BYTE(SIZEOF(CTRL2));
CTRL3._CTRL8.SIZE:=ANY_TO_BYTE(SIZEOF(CTRL3));
TIMER(IN:=TRUE, PT:=T#500mS);
IF	TIMER.Q THEN
	TIMER(IN:=FALSE);
	CASE STAGE OF
		0:
			SET_BIT8(ADR(CTRL2),N);
			AND8(ADR(CTRL1),ADR(CTRL2),ADR(CTRL3));
			X1 := GET_BIT8(ADR(CTRL1),N);
			X2 := GET_BIT8(ADR(CTRL2),N);
			X3 := GET_BIT8(ADR(CTRL3),N);
			STAGE := 1;
		1:
			RESET_BIT8(ADR(CTRL2),N);
			SET_BIT8(ADR(CTRL1),N);
			AND8(ADR(CTRL1),ADR(CTRL2),ADR(CTRL3));
			X1 := GET_BIT8(ADR(CTRL1),N);
			X2 := GET_BIT8(ADR(CTRL2),N);
			X3 := GET_BIT8(ADR(CTRL3),N);
			STAGE := 2;
		2:
			SET_BIT8(ADR(CTRL2),N);
			AND8(ADR(CTRL1),ADR(CTRL2),ADR(CTRL3));
			X1 := GET_BIT8(ADR(CTRL1),N);
			X2 := GET_BIT8(ADR(CTRL2),N);
			X3 := GET_BIT8(ADR(CTRL3),N);
			STAGE := 3;
		3:
			RESET_BIT8(ADR(CTRL1),N);
			RESET_BIT8(ADR(CTRL2),N);
			AND8(ADR(CTRL1),ADR(CTRL2),ADR(CTRL3));
			X1 := GET_BIT8(ADR(CTRL1),N);
			X2 := GET_BIT8(ADR(CTRL2),N);
			X3 := GET_BIT8(ADR(CTRL3),N);
			STAGE := 0;
			N:=N+1;
			IF	N = 16 THEN
				N := 0;
			END_IF
	END_CASE
END_IF
IF	X3 = (X1 AND X2) THEN
	CORRECT	:=	TRUE;
ELSE
	CORRECT	:=	FALSE;
END_IF
          
END_PROGRAM

PROGRAM CHECK_AND16
  VAR
    CTRL1 : uCTRL16;
    CTRL2 : uCTRL16;
    CTRL3 : uCTRL16;
    TIMER : TON;
    STAGE : ENUM;
    N : LINT;
    X1 : BOOL;
    X2 : BOOL;
    X3 : BOOL;
    CORRECT : BOOL := TRUE;
  END_VAR

            CTRL1._CTRL16.SIZE:=ANY_TO_WORD(SIZEOF(CTRL1));
CTRL2._CTRL16.SIZE:=ANY_TO_WORD(SIZEOF(CTRL2));
CTRL3._CTRL16.SIZE:=ANY_TO_WORD(SIZEOF(CTRL3));
TIMER(IN:=TRUE, PT:=T#500MS);
IF	TIMER.Q THEN
	TIMER(IN:=FALSE);
	CASE STAGE OF
		0:
			SET_BIT16(ADR(CTRL2),N);
			AND16(ADR(CTRL1),ADR(CTRL2),ADR(CTRL3));
			X1 := GET_BIT16(ADR(CTRL1),N);
			X2 := GET_BIT16(ADR(CTRL2),N);
			X3 := GET_BIT16(ADR(CTRL3),N);
			STAGE := 1;
		1:
			RESET_BIT16(ADR(CTRL2),N);
			SET_BIT16(ADR(CTRL1),N);
			AND16(ADR(CTRL1),ADR(CTRL2),ADR(CTRL3));
			X1 := GET_BIT16(ADR(CTRL1),N);
			X2 := GET_BIT16(ADR(CTRL2),N);
			X3 := GET_BIT16(ADR(CTRL3),N);
			STAGE := 2;
		2:
			SET_BIT16(ADR(CTRL2),N);
			AND16(ADR(CTRL1),ADR(CTRL2),ADR(CTRL3));
			X1 := GET_BIT16(ADR(CTRL1),N);
			X2 := GET_BIT16(ADR(CTRL2),N);
			X3 := GET_BIT16(ADR(CTRL3),N);
			STAGE := 3;
		3:
			RESET_BIT16(ADR(CTRL1),N);
			RESET_BIT16(ADR(CTRL2),N);
			AND16(ADR(CTRL1),ADR(CTRL2),ADR(CTRL3));
			X1 := GET_BIT16(ADR(CTRL1),N);
			X2 := GET_BIT16(ADR(CTRL2),N);
			X3 := GET_BIT16(ADR(CTRL3),N);
			STAGE := 0;
			N:=N+1;
			IF	N = 32 THEN
				N := 0;
			END_IF
	END_CASE
END_IF
IF	X3 = (X1 AND X2) THEN
	CORRECT	:=	TRUE;
ELSE
	CORRECT	:=	FALSE;
END_IF
          
END_PROGRAM

PROGRAM CHECK_AND32
  VAR
    CTRL1 : uCTRL32;
    CTRL2 : uCTRL32;
    CTRL3 : uCTRL32;
    TIMER : TON;
    STAGE : ENUM;
    N : LINT;
    X1 : BOOL;
    X2 : BOOL;
    X3 : BOOL;
    CORRECT : BOOL := TRUE;
  END_VAR

            CTRL1._CTRL32.SIZE:=ANY_TO_DWORD(SIZEOF(CTRL1));
CTRL2._CTRL32.SIZE:=ANY_TO_DWORD(SIZEOF(CTRL2));
CTRL3._CTRL32.SIZE:=ANY_TO_DWORD(SIZEOF(CTRL3));
TIMER(IN:=TRUE, PT:=T#500MS);
IF	TIMER.Q THEN
	TIMER(IN:=FALSE);
	CASE STAGE OF
		0:
			SET_BIT32(ADR(CTRL2),N);
			AND32(ADR(CTRL1),ADR(CTRL2),ADR(CTRL3));
			X1 := GET_BIT32(ADR(CTRL1),N);
			X2 := GET_BIT32(ADR(CTRL2),N);
			X3 := GET_BIT32(ADR(CTRL3),N);
			STAGE := 1;
		1:
			RESET_BIT32(ADR(CTRL2),N);
			SET_BIT32(ADR(CTRL1),N);
			AND32(ADR(CTRL1),ADR(CTRL2),ADR(CTRL3));
			X1 := GET_BIT32(ADR(CTRL1),N);
			X2 := GET_BIT32(ADR(CTRL2),N);
			X3 := GET_BIT32(ADR(CTRL3),N);
			STAGE := 2;
		2:
			SET_BIT32(ADR(CTRL2),N);
			AND32(ADR(CTRL1),ADR(CTRL2),ADR(CTRL3));
			X1 := GET_BIT32(ADR(CTRL1),N);
			X2 := GET_BIT32(ADR(CTRL2),N);
			X3 := GET_BIT32(ADR(CTRL3),N);
			STAGE := 3;
		3:
			RESET_BIT32(ADR(CTRL1),N);
			RESET_BIT32(ADR(CTRL2),N);
			AND32(ADR(CTRL1),ADR(CTRL2),ADR(CTRL3));
			X1 := GET_BIT32(ADR(CTRL1),N);
			X2 := GET_BIT32(ADR(CTRL2),N);
			X3 := GET_BIT32(ADR(CTRL3),N);
			STAGE := 0;
			N:=N+1;
			IF	N = 64 THEN
				N := 0;
			END_IF
	END_CASE
END_IF
IF	X3 = (X1 AND X2) THEN
	CORRECT	:=	TRUE;
ELSE
	CORRECT	:=	FALSE;
END_IF
          
END_PROGRAM

PROGRAM CHECK_EQ8
  VAR
    CTRL1 : uCTRL8;
    CTRL2 : uCTRL8;
    CTRL3 : uCTRL8;
    TIMER : TON;
    STAGE : ENUM;
    N : LINT;
    X1 : BOOL;
    X2 : BOOL;
    X3 : BOOL;
    CORRECT : BOOL := TRUE;
  END_VAR

            CTRL1._CTRL8.SIZE:=ANY_TO_BYTE(SIZEOF(CTRL1));
CTRL2._CTRL8.SIZE:=ANY_TO_BYTE(SIZEOF(CTRL2));
CTRL3._CTRL8.SIZE:=ANY_TO_BYTE(SIZEOF(CTRL3));
TIMER(IN:=TRUE, PT:=T#500mS);
IF	TIMER.Q THEN
	TIMER(IN:=FALSE);
	CASE STAGE OF
		0:
			SET_BIT8(ADR(CTRL2),N);
			EQ8(ADR(CTRL1),ADR(CTRL2),ADR(CTRL3));
			X1 := GET_BIT8(ADR(CTRL1),N);
			X2 := GET_BIT8(ADR(CTRL2),N);
			X3 := GET_BIT8(ADR(CTRL3),N);
			STAGE := 1;
		1:
			RESET_BIT8(ADR(CTRL2),N);
			SET_BIT8(ADR(CTRL1),N);
			EQ8(ADR(CTRL1),ADR(CTRL2),ADR(CTRL3));
			X1 := GET_BIT8(ADR(CTRL1),N);
			X2 := GET_BIT8(ADR(CTRL2),N);
			X3 := GET_BIT8(ADR(CTRL3),N);
			STAGE := 2;
		2:
			SET_BIT8(ADR(CTRL2),N);
			EQ8(ADR(CTRL1),ADR(CTRL2),ADR(CTRL3));
			X1 := GET_BIT8(ADR(CTRL1),N);
			X2 := GET_BIT8(ADR(CTRL2),N);
			X3 := GET_BIT8(ADR(CTRL3),N);
			STAGE := 3;
		3:
			RESET_BIT8(ADR(CTRL1),N);
			RESET_BIT8(ADR(CTRL2),N);
			EQ8(ADR(CTRL1),ADR(CTRL2),ADR(CTRL3));
			X1 := GET_BIT8(ADR(CTRL1),N);
			X2 := GET_BIT8(ADR(CTRL2),N);
			X3 := GET_BIT8(ADR(CTRL3),N);
			STAGE := 0;
			N:=N+1;
			IF	N = 16 THEN
				N := 0;
			END_IF
	END_CASE
END_IF
IF	X3 = (X1 = X2) THEN
	CORRECT	:=	TRUE;
ELSE
	CORRECT	:=	FALSE;
END_IF
          
END_PROGRAM

PROGRAM CHECK_EQ16
  VAR
    CTRL1 : uCTRL16;
    CTRL2 : uCTRL16;
    CTRL3 : uCTRL16;
    TIMER : TON;
    STAGE : ENUM;
    N : LINT;
    X1 : BOOL;
    X2 : BOOL;
    X3 : BOOL;
    CORRECT : BOOL := TRUE;
  END_VAR

            CTRL1._CTRL16.SIZE:=ANY_TO_WORD(SIZEOF(CTRL1));
CTRL2._CTRL16.SIZE:=ANY_TO_WORD(SIZEOF(CTRL2));
CTRL3._CTRL16.SIZE:=ANY_TO_WORD(SIZEOF(CTRL3));
TIMER(IN:=TRUE, PT:=T#500MS);
IF	TIMER.Q THEN
	TIMER(IN:=FALSE);
	CASE STAGE OF
		0:
			SET_BIT16(ADR(CTRL2),N);
			EQ16(ADR(CTRL1),ADR(CTRL2),ADR(CTRL3));
			X1 := GET_BIT16(ADR(CTRL1),N);
			X2 := GET_BIT16(ADR(CTRL2),N);
			X3 := GET_BIT16(ADR(CTRL3),N);
			STAGE := 1;
		1:
			RESET_BIT16(ADR(CTRL2),N);
			SET_BIT16(ADR(CTRL1),N);
			EQ16(ADR(CTRL1),ADR(CTRL2),ADR(CTRL3));
			X1 := GET_BIT16(ADR(CTRL1),N);
			X2 := GET_BIT16(ADR(CTRL2),N);
			X3 := GET_BIT16(ADR(CTRL3),N);
			STAGE := 2;
		2:
			SET_BIT16(ADR(CTRL2),N);
			EQ16(ADR(CTRL1),ADR(CTRL2),ADR(CTRL3));
			X1 := GET_BIT16(ADR(CTRL1),N);
			X2 := GET_BIT16(ADR(CTRL2),N);
			X3 := GET_BIT16(ADR(CTRL3),N);
			STAGE := 3;
		3:
			RESET_BIT16(ADR(CTRL1),N);
			RESET_BIT16(ADR(CTRL2),N);
			EQ16(ADR(CTRL1),ADR(CTRL2),ADR(CTRL3));
			X1 := GET_BIT16(ADR(CTRL1),N);
			X2 := GET_BIT16(ADR(CTRL2),N);
			X3 := GET_BIT16(ADR(CTRL3),N);
			STAGE := 0;
			N:=N+1;
			IF	N = 32 THEN
				N := 0;
			END_IF
	END_CASE
END_IF
IF	X3 = (X1 = X2) THEN
	CORRECT	:=	TRUE;
ELSE
	CORRECT	:=	FALSE;
END_IF
          
END_PROGRAM

PROGRAM CHECK_EQ32
  VAR
    CTRL1 : uCTRL32;
    CTRL2 : uCTRL32;
    CTRL3 : uCTRL32;
    TIMER : TON;
    STAGE : ENUM;
    N : LINT;
    X1 : BOOL;
    X2 : BOOL;
    X3 : BOOL;
    CORRECT : BOOL := TRUE;
  END_VAR

            CTRL1._CTRL32.SIZE:=ANY_TO_DWORD(SIZEOF(CTRL1));
CTRL2._CTRL32.SIZE:=ANY_TO_DWORD(SIZEOF(CTRL2));
CTRL3._CTRL32.SIZE:=ANY_TO_DWORD(SIZEOF(CTRL3));
TIMER(IN:=TRUE, PT:=T#500MS);
IF	TIMER.Q THEN
	TIMER(IN:=FALSE);
	CASE STAGE OF
		0:
			SET_BIT32(ADR(CTRL2),N);
			EQ32(ADR(CTRL1),ADR(CTRL2),ADR(CTRL3));
			X1 := GET_BIT32(ADR(CTRL1),N);
			X2 := GET_BIT32(ADR(CTRL2),N);
			X3 := GET_BIT32(ADR(CTRL3),N);
			STAGE := 1;
		1:
			RESET_BIT32(ADR(CTRL2),N);
			SET_BIT32(ADR(CTRL1),N);
			EQ32(ADR(CTRL1),ADR(CTRL2),ADR(CTRL3));
			X1 := GET_BIT32(ADR(CTRL1),N);
			X2 := GET_BIT32(ADR(CTRL2),N);
			X3 := GET_BIT32(ADR(CTRL3),N);
			STAGE := 2;
		2:
			SET_BIT32(ADR(CTRL2),N);
			EQ32(ADR(CTRL1),ADR(CTRL2),ADR(CTRL3));
			X1 := GET_BIT32(ADR(CTRL1),N);
			X2 := GET_BIT32(ADR(CTRL2),N);
			X3 := GET_BIT32(ADR(CTRL3),N);
			STAGE := 3;
		3:
			RESET_BIT32(ADR(CTRL1),N);
			RESET_BIT32(ADR(CTRL2),N);
			EQ32(ADR(CTRL1),ADR(CTRL2),ADR(CTRL3));
			X1 := GET_BIT32(ADR(CTRL1),N);
			X2 := GET_BIT32(ADR(CTRL2),N);
			X3 := GET_BIT32(ADR(CTRL3),N);
			STAGE := 0;
			N:=N+1;
			IF	N = 64 THEN
				N := 0;
			END_IF
	END_CASE
END_IF
IF	X3 = (X1 = X2) THEN
	CORRECT	:=	TRUE;
ELSE
	CORRECT	:=	FALSE;
END_IF
          
END_PROGRAM

PROGRAM CHECK_NAND8
  VAR
    CTRL1 : uCTRL8;
    CTRL2 : uCTRL8;
    CTRL3 : uCTRL8;
    TIMER : TON;
    STAGE : ENUM;
    N : LINT;
    X1 : BOOL;
    X2 : BOOL;
    X3 : BOOL;
    CORRECT : BOOL := TRUE;
  END_VAR

            CTRL1._CTRL8.SIZE:=ANY_TO_BYTE(SIZEOF(CTRL1));
CTRL2._CTRL8.SIZE:=ANY_TO_BYTE(SIZEOF(CTRL2));
CTRL3._CTRL8.SIZE:=ANY_TO_BYTE(SIZEOF(CTRL3));
TIMER(IN:=TRUE, PT:=T#500mS);
IF	TIMER.Q THEN
	TIMER(IN:=FALSE);
	CASE STAGE OF
		0:
			SET_BIT8(ADR(CTRL2),N);
			NAND8(ADR(CTRL1),ADR(CTRL2),ADR(CTRL3));
			X1 := GET_BIT8(ADR(CTRL1),N);
			X2 := GET_BIT8(ADR(CTRL2),N);
			X3 := GET_BIT8(ADR(CTRL3),N);
			STAGE := 1;
		1:
			RESET_BIT8(ADR(CTRL2),N);
			SET_BIT8(ADR(CTRL1),N);
			NAND8(ADR(CTRL1),ADR(CTRL2),ADR(CTRL3));
			X1 := GET_BIT8(ADR(CTRL1),N);
			X2 := GET_BIT8(ADR(CTRL2),N);
			X3 := GET_BIT8(ADR(CTRL3),N);
			STAGE := 2;
		2:
			SET_BIT8(ADR(CTRL2),N);
			NAND8(ADR(CTRL1),ADR(CTRL2),ADR(CTRL3));
			X1 := GET_BIT8(ADR(CTRL1),N);
			X2 := GET_BIT8(ADR(CTRL2),N);
			X3 := GET_BIT8(ADR(CTRL3),N);
			STAGE := 3;
		3:
			RESET_BIT8(ADR(CTRL1),N);
			RESET_BIT8(ADR(CTRL2),N);
			NAND8(ADR(CTRL1),ADR(CTRL2),ADR(CTRL3));
			X1 := GET_BIT8(ADR(CTRL1),N);
			X2 := GET_BIT8(ADR(CTRL2),N);
			X3 := GET_BIT8(ADR(CTRL3),N);
			STAGE := 0;
			N:=N+1;
			IF	N = 16 THEN
				N := 0;
			END_IF
	END_CASE
END_IF
IF	X3 = NOT(X1 AND X2) THEN
	CORRECT	:=	TRUE;
ELSE
	CORRECT	:=	FALSE;
END_IF
          
END_PROGRAM

PROGRAM CHECK_NAND16
  VAR
    CTRL1 : uCTRL16;
    CTRL2 : uCTRL16;
    CTRL3 : uCTRL16;
    TIMER : TON;
    STAGE : ENUM;
    N : LINT;
    X1 : BOOL;
    X2 : BOOL;
    X3 : BOOL;
    CORRECT : BOOL := TRUE;
  END_VAR

            CTRL1._CTRL16.SIZE:=ANY_TO_WORD(SIZEOF(CTRL1));
CTRL2._CTRL16.SIZE:=ANY_TO_WORD(SIZEOF(CTRL2));
CTRL3._CTRL16.SIZE:=ANY_TO_WORD(SIZEOF(CTRL3));
TIMER(IN:=TRUE, PT:=T#500MS);
IF	TIMER.Q THEN
	TIMER(IN:=FALSE);
	CASE STAGE OF
		0:
			SET_BIT16(ADR(CTRL2),N);
			NAND16(ADR(CTRL1),ADR(CTRL2),ADR(CTRL3));
			X1 := GET_BIT16(ADR(CTRL1),N);
			X2 := GET_BIT16(ADR(CTRL2),N);
			X3 := GET_BIT16(ADR(CTRL3),N);
			STAGE := 1;
		1:
			RESET_BIT16(ADR(CTRL2),N);
			SET_BIT16(ADR(CTRL1),N);
			NAND16(ADR(CTRL1),ADR(CTRL2),ADR(CTRL3));
			X1 := GET_BIT16(ADR(CTRL1),N);
			X2 := GET_BIT16(ADR(CTRL2),N);
			X3 := GET_BIT16(ADR(CTRL3),N);
			STAGE := 2;
		2:
			SET_BIT16(ADR(CTRL2),N);
			NAND16(ADR(CTRL1),ADR(CTRL2),ADR(CTRL3));
			X1 := GET_BIT16(ADR(CTRL1),N);
			X2 := GET_BIT16(ADR(CTRL2),N);
			X3 := GET_BIT16(ADR(CTRL3),N);
			STAGE := 3;
		3:
			RESET_BIT16(ADR(CTRL1),N);
			RESET_BIT16(ADR(CTRL2),N);
			NAND16(ADR(CTRL1),ADR(CTRL2),ADR(CTRL3));
			X1 := GET_BIT16(ADR(CTRL1),N);
			X2 := GET_BIT16(ADR(CTRL2),N);
			X3 := GET_BIT16(ADR(CTRL3),N);
			STAGE := 0;
			N:=N+1;
			IF	N = 32 THEN
				N := 0;
			END_IF
	END_CASE
END_IF
IF	X3 = NOT(X1 AND X2) THEN
	CORRECT	:=	TRUE;
ELSE
	CORRECT	:=	FALSE;
END_IF
          
END_PROGRAM

PROGRAM CHECK_NAND32
  VAR
    CTRL1 : uCTRL32;
    CTRL2 : uCTRL32;
    CTRL3 : uCTRL32;
    TIMER : TON;
    STAGE : ENUM;
    N : LINT;
    X1 : BOOL;
    X2 : BOOL;
    X3 : BOOL;
    CORRECT : BOOL := TRUE;
  END_VAR

            CTRL1._CTRL32.SIZE:=ANY_TO_DWORD(SIZEOF(CTRL1));
CTRL2._CTRL32.SIZE:=ANY_TO_DWORD(SIZEOF(CTRL2));
CTRL3._CTRL32.SIZE:=ANY_TO_DWORD(SIZEOF(CTRL3));
TIMER(IN:=TRUE, PT:=T#500MS);
IF	TIMER.Q THEN
	TIMER(IN:=FALSE);
	CASE STAGE OF
		0:
			SET_BIT32(ADR(CTRL2),N);
			NAND32(ADR(CTRL1),ADR(CTRL2),ADR(CTRL3));
			X1 := GET_BIT32(ADR(CTRL1),N);
			X2 := GET_BIT32(ADR(CTRL2),N);
			X3 := GET_BIT32(ADR(CTRL3),N);
			STAGE := 1;
		1:
			RESET_BIT32(ADR(CTRL2),N);
			SET_BIT32(ADR(CTRL1),N);
			NAND32(ADR(CTRL1),ADR(CTRL2),ADR(CTRL3));
			X1 := GET_BIT32(ADR(CTRL1),N);
			X2 := GET_BIT32(ADR(CTRL2),N);
			X3 := GET_BIT32(ADR(CTRL3),N);
			STAGE := 2;
		2:
			SET_BIT32(ADR(CTRL2),N);
			NAND32(ADR(CTRL1),ADR(CTRL2),ADR(CTRL3));
			X1 := GET_BIT32(ADR(CTRL1),N);
			X2 := GET_BIT32(ADR(CTRL2),N);
			X3 := GET_BIT32(ADR(CTRL3),N);
			STAGE := 3;
		3:
			RESET_BIT32(ADR(CTRL1),N);
			RESET_BIT32(ADR(CTRL2),N);
			NAND32(ADR(CTRL1),ADR(CTRL2),ADR(CTRL3));
			X1 := GET_BIT32(ADR(CTRL1),N);
			X2 := GET_BIT32(ADR(CTRL2),N);
			X3 := GET_BIT32(ADR(CTRL3),N);
			STAGE := 0;
			N:=N+1;
			IF	N = 64 THEN
				N := 0;
			END_IF
	END_CASE
END_IF
IF	X3 = NOT(X1 AND X2) THEN
	CORRECT	:=	TRUE;
ELSE
	CORRECT	:=	FALSE;
END_IF
          
END_PROGRAM

PROGRAM CHECK_NEQ8
  VAR
    CTRL1 : uCTRL8;
    CTRL2 : uCTRL8;
    CTRL3 : uCTRL8;
    TIMER : TON;
    STAGE : ENUM;
    N : LINT;
    X1 : BOOL;
    X2 : BOOL;
    X3 : BOOL;
    CORRECT : BOOL := TRUE;
  END_VAR

            CTRL1._CTRL8.SIZE:=ANY_TO_BYTE(SIZEOF(CTRL1));
CTRL2._CTRL8.SIZE:=ANY_TO_BYTE(SIZEOF(CTRL2));
CTRL3._CTRL8.SIZE:=ANY_TO_BYTE(SIZEOF(CTRL3));
TIMER(IN:=TRUE, PT:=T#500mS);
IF	TIMER.Q THEN
	TIMER(IN:=FALSE);
	CASE STAGE OF
		0:
			SET_BIT8(ADR(CTRL2),N);
			NEQ8(ADR(CTRL1),ADR(CTRL2),ADR(CTRL3));
			X1 := GET_BIT8(ADR(CTRL1),N);
			X2 := GET_BIT8(ADR(CTRL2),N);
			X3 := GET_BIT8(ADR(CTRL3),N);
			STAGE := 1;
		1:
			RESET_BIT8(ADR(CTRL2),N);
			SET_BIT8(ADR(CTRL1),N);
			NEQ8(ADR(CTRL1),ADR(CTRL2),ADR(CTRL3));
			X1 := GET_BIT8(ADR(CTRL1),N);
			X2 := GET_BIT8(ADR(CTRL2),N);
			X3 := GET_BIT8(ADR(CTRL3),N);
			STAGE := 2;
		2:
			SET_BIT8(ADR(CTRL2),N);
			NEQ8(ADR(CTRL1),ADR(CTRL2),ADR(CTRL3));
			X1 := GET_BIT8(ADR(CTRL1),N);
			X2 := GET_BIT8(ADR(CTRL2),N);
			X3 := GET_BIT8(ADR(CTRL3),N);
			STAGE := 3;
		3:
			RESET_BIT8(ADR(CTRL1),N);
			RESET_BIT8(ADR(CTRL2),N);
			NEQ8(ADR(CTRL1),ADR(CTRL2),ADR(CTRL3));
			X1 := GET_BIT8(ADR(CTRL1),N);
			X2 := GET_BIT8(ADR(CTRL2),N);
			X3 := GET_BIT8(ADR(CTRL3),N);
			STAGE := 0;
			N:=N+1;
			IF	N = 16 THEN
				N := 0;
			END_IF
	END_CASE
END_IF
IF	X3 = NOT(X1 = X2) THEN
	CORRECT	:=	TRUE;
ELSE
	CORRECT	:=	FALSE;
END_IF
          
END_PROGRAM

PROGRAM CHECK_NEQ16
  VAR
    CTRL1 : uCTRL16;
    CTRL2 : uCTRL16;
    CTRL3 : uCTRL16;
    TIMER : TON;
    STAGE : ENUM;
    N : LINT;
    X1 : BOOL;
    X2 : BOOL;
    X3 : BOOL;
    CORRECT : BOOL := TRUE;
  END_VAR

            CTRL1._CTRL16.SIZE:=ANY_TO_WORD(SIZEOF(CTRL1));
CTRL2._CTRL16.SIZE:=ANY_TO_WORD(SIZEOF(CTRL2));
CTRL3._CTRL16.SIZE:=ANY_TO_WORD(SIZEOF(CTRL3));
TIMER(IN:=TRUE, PT:=T#500MS);
IF	TIMER.Q THEN
	TIMER(IN:=FALSE);
	CASE STAGE OF
		0:
			SET_BIT16(ADR(CTRL2),N);
			NEQ16(ADR(CTRL1),ADR(CTRL2),ADR(CTRL3));
			X1 := GET_BIT16(ADR(CTRL1),N);
			X2 := GET_BIT16(ADR(CTRL2),N);
			X3 := GET_BIT16(ADR(CTRL3),N);
			STAGE := 1;
		1:
			RESET_BIT16(ADR(CTRL2),N);
			SET_BIT16(ADR(CTRL1),N);
			NEQ16(ADR(CTRL1),ADR(CTRL2),ADR(CTRL3));
			X1 := GET_BIT16(ADR(CTRL1),N);
			X2 := GET_BIT16(ADR(CTRL2),N);
			X3 := GET_BIT16(ADR(CTRL3),N);
			STAGE := 2;
		2:
			SET_BIT16(ADR(CTRL2),N);
			NEQ16(ADR(CTRL1),ADR(CTRL2),ADR(CTRL3));
			X1 := GET_BIT16(ADR(CTRL1),N);
			X2 := GET_BIT16(ADR(CTRL2),N);
			X3 := GET_BIT16(ADR(CTRL3),N);
			STAGE := 3;
		3:
			RESET_BIT16(ADR(CTRL1),N);
			RESET_BIT16(ADR(CTRL2),N);
			NEQ16(ADR(CTRL1),ADR(CTRL2),ADR(CTRL3));
			X1 := GET_BIT16(ADR(CTRL1),N);
			X2 := GET_BIT16(ADR(CTRL2),N);
			X3 := GET_BIT16(ADR(CTRL3),N);
			STAGE := 0;
			N:=N+1;
			IF	N = 32 THEN
				N := 0;
			END_IF
	END_CASE
END_IF
IF	X3 = NOT(X1 = X2) THEN
	CORRECT	:=	TRUE;
ELSE
	CORRECT	:=	FALSE;
END_IF
          
END_PROGRAM

PROGRAM CHECK_FIND1ST_1_8
  VAR
    CTRL1 : uCTRL8;
    N : LINT;
  END_VAR

            CTRL1._CTRL8.SIZE:=ANY_TO_BYTE(SIZEOF(CTRL1));
N:=FIND1ST_1_8(ADR(CTRL1));
          
END_PROGRAM

PROGRAM CHECK_FIND1ST_1_32
  VAR
    CTRL1 : uCTRL32;
    N : LINT;
  END_VAR

            CTRL1._CTRL32.SIZE:=ANY_TO_DWORD(SIZEOF(CTRL1));
N:=FIND1ST_1_32(ADR(CTRL1));
          
END_PROGRAM

PROGRAM CHECK_FIND1ST_0_8
  VAR
    CTRL1 : uCTRL8;
    N : LINT;
  END_VAR

            CTRL1._CTRL8.SIZE:=ANY_TO_BYTE(SIZEOF(CTRL1));
N:=FIND1ST_0_8(ADR(CTRL1));
          
END_PROGRAM

PROGRAM CHECK_FIND1ST_0_16
  VAR
    CTRL1 : uCTRL16;
    N : LINT;
  END_VAR

            CTRL1._CTRL16.SIZE:=ANY_TO_WORD(SIZEOF(CTRL1));
N:=FIND1ST_0_16(ADR(CTRL1));
          
END_PROGRAM

PROGRAM CHECK_FIND1ST_0_32
  VAR
    CTRL1 : uCTRL32;
    N : LINT;
  END_VAR

            CTRL1._CTRL32.SIZE:=ANY_TO_DWORD(SIZEOF(CTRL1));
N:=FIND1ST_0_32(ADR(CTRL1));
          
END_PROGRAM

PROGRAM CHECK_SET_BIT16
  VAR
    CTRL1 : uCTRL16;
    N : LINT;
  END_VAR

            CTRL1._CTRL16.SIZE:=ANY_TO_WORD(SIZEOF(CTRL1));
SET_BIT16(ADR(CTRL1),N,);
          
END_PROGRAM

PROGRAM CHECK_SET_BIT8
  VAR
    CTRL1 : uCTRL8;
    N : LINT;
  END_VAR

            CTRL1._CTRL8.SIZE:=ANY_TO_BYTE(SIZEOF(CTRL1));
SET_BIT8(ADR(CTRL1),N);
          
END_PROGRAM

PROGRAM CHECK_SET_BIT32
  VAR
    CTRL1 : uCTRL32;
    N : LINT;
  END_VAR

            CTRL1._CTRL32.SIZE:=ANY_TO_DWORD(SIZEOF(CTRL1));
SET_BIT32(ADR(CTRL1),N);
          
END_PROGRAM

PROGRAM CHECK_RESET_BIT16
  VAR
    CTRL1 : uCTRL16;
    N : LINT;
  END_VAR

            CTRL1._CTRL16.SIZE:=ANY_TO_WORD(SIZEOF(CTRL1));
RESET_BIT16(ADR(CTRL1),N);
          
END_PROGRAM

PROGRAM CHECK_RESET_BIT32
  VAR
    CTRL1 : uCTRL32;
    N : LINT;
  END_VAR

            CTRL1._CTRL32.SIZE:=ANY_TO_DWORD(SIZEOF(CTRL1));
RESET_BIT32(ADR(CTRL1),N);
          
END_PROGRAM

PROGRAM CHECK_RESET_BIT8
  VAR
    CTRL1 : uCTRL8;
    N : LINT;
  END_VAR

            CTRL1._CTRL8.SIZE:=ANY_TO_BYTE(SIZEOF(CTRL1));
RESET_BIT8(ADR(CTRL1),N);
          
END_PROGRAM

FUNCTION RESET_BIT16 : BOOL
  VAR_INPUT
    IN_ADR : POINTER TO WORD;
    BIT_NUMBER : LINT;
  END_VAR
  VAR
    SIZE : WORD;
    pwADR : POINTER TO WORD;
    wWORD : WORD;
  END_VAR
  VAR CONSTANT
    STEP : WORD := 2;
    STEP_SIZE : WORD := (STEP * 8);
  END_VAR

            pwADR:=	IN_ADR+STEP;
SIZE	:=	pwADR^;	
IF BIT_NUMBER >= (SIZE-2*STEP)*8 OR BIT_NUMBER <0 THEN
	BIT_NUMBER	:=	0;
	BIT_NUMBER	:=	BIT_NUMBER/BIT_NUMBER;
	//Ты вышел за пределы структуры, дядь
END_IF
pwADR := IN_ADR + (2 + ANY_TO_DWORD(BIT_NUMBER/STEP_SIZE))*STEP;
wWORD:=NOT(SHL(1,BIT_NUMBER MOD STEP_SIZE));
pwADR^ := pwADR^ AND wWORD;
          
END_FUNCTION

FUNCTION RESET_BIT32 : BOOL
  VAR_INPUT
    IN_ADR : POINTER TO DWORD;
    BIT_NUMBER : LINT;
  END_VAR
  VAR
    SIZE : DWORD;
    pdwADR : POINTER TO DWORD;
    dwDWORD : DWORD;
  END_VAR
  VAR CONSTANT
    STEP : WORD := 4;
    STEP_SIZE : WORD := (STEP * 8);
  END_VAR

            pdwADR:=	IN_ADR+STEP;
SIZE	:=	pdwADR^;	
IF BIT_NUMBER >= (SIZE-2*STEP)*8 OR BIT_NUMBER <0 THEN
	BIT_NUMBER	:=	0;
	BIT_NUMBER	:=	BIT_NUMBER/BIT_NUMBER;
	//Ты вышел за пределы структуры, дядь
END_IF
pdwADR := IN_ADR + (2 + ANY_TO_DWORD(BIT_NUMBER/STEP_SIZE))*STEP;
dwDWORD:=NOT(SHL(1,BIT_NUMBER MOD STEP_SIZE));
pdwADR^ := pdwADR^ AND dwDWORD;
          
END_FUNCTION

FUNCTION RESET_BIT8 : BOOL
  VAR_INPUT
    IN_ADR : POINTER TO BYTE;
    BIT_NUMBER : LINT;
  END_VAR
  VAR
    SIZE : BYTE;
    pbADR : POINTER TO BYTE;
    bBYTE : BYTE;
  END_VAR
  VAR CONSTANT
    STEP : BYTE := 1;
    STEP_SIZE : BYTE := (STEP * 8);
  END_VAR

            pbADR:=	IN_ADR+STEP;
SIZE	:=	pbADR^;	
IF BIT_NUMBER >= (SIZE-2*STEP)*8 OR BIT_NUMBER <0 THEN
	BIT_NUMBER	:=	0;
	BIT_NUMBER	:=	BIT_NUMBER/BIT_NUMBER;
	//Ты вышел за пределы структуры, дядь
END_IF
pbADR := IN_ADR + 2*STEP + ANY_TO_DWORD(BIT_NUMBER/STEP_SIZE);
bBYTE:=NOT(SHL(1,BIT_NUMBER MOD STEP_SIZE));
pbADR^ := pbADR^ AND bBYTE;
          
END_FUNCTION

PROGRAM CHECK_OR8
  VAR
    CTRL1 : uCTRL8;
    CTRL2 : uCTRL8;
    CTRL3 : uCTRL8;
    TIMER : TON;
    STAGE : ENUM;
    N : LINT;
    X1 : BOOL;
    X2 : BOOL;
    X3 : BOOL;
    CORRECT : BOOL := TRUE;
  END_VAR

            CTRL1._CTRL8.SIZE:=ANY_TO_BYTE(SIZEOF(CTRL1));
CTRL2._CTRL8.SIZE:=ANY_TO_BYTE(SIZEOF(CTRL2));
CTRL3._CTRL8.SIZE:=ANY_TO_BYTE(SIZEOF(CTRL3));
TIMER(IN:=TRUE, PT:=T#500mS);
IF	TIMER.Q THEN
	TIMER(IN:=FALSE);
	CASE STAGE OF
		0:
			SET_BIT8(ADR(CTRL2),N);
			OR8(ADR(CTRL1),ADR(CTRL2),ADR(CTRL3));
			X1 := GET_BIT8(ADR(CTRL1),N);
			X2 := GET_BIT8(ADR(CTRL2),N);
			X3 := GET_BIT8(ADR(CTRL3),N);
			STAGE := 1;
		1:
			RESET_BIT8(ADR(CTRL2),N);
			SET_BIT8(ADR(CTRL1),N);
			OR8(ADR(CTRL1),ADR(CTRL2),ADR(CTRL3));
			X1 := GET_BIT8(ADR(CTRL1),N);
			X2 := GET_BIT8(ADR(CTRL2),N);
			X3 := GET_BIT8(ADR(CTRL3),N);
			STAGE := 2;
		2:
			SET_BIT8(ADR(CTRL2),N);
			OR8(ADR(CTRL1),ADR(CTRL2),ADR(CTRL3));
			X1 := GET_BIT8(ADR(CTRL1),N);
			X2 := GET_BIT8(ADR(CTRL2),N);
			X3 := GET_BIT8(ADR(CTRL3),N);
			STAGE := 3;
		3:
			RESET_BIT8(ADR(CTRL1),N);
			RESET_BIT8(ADR(CTRL2),N);
			OR8(ADR(CTRL1),ADR(CTRL2),ADR(CTRL3));
			X1 := GET_BIT8(ADR(CTRL1),N);
			X2 := GET_BIT8(ADR(CTRL2),N);
			X3 := GET_BIT8(ADR(CTRL3),N);
			STAGE := 0;
			N:=N+1;
			IF	N = 16 THEN
				N := 0;
			END_IF
	END_CASE
END_IF
IF	X3 = (X1 OR X2) THEN
	CORRECT	:=	TRUE;
ELSE
	CORRECT	:=	FALSE;
END_IF
          
END_PROGRAM

PROGRAM CHECK_OR16
  VAR
    CTRL1 : uCTRL16;
    CTRL2 : uCTRL16;
    CTRL3 : uCTRL16;
    TIMER : TON;
    STAGE : ENUM;
    N : LINT;
    X1 : BOOL;
    X2 : BOOL;
    X3 : BOOL;
    CORRECT : BOOL := TRUE;
  END_VAR

            CTRL1._CTRL16.SIZE:=ANY_TO_WORD(SIZEOF(CTRL1));
CTRL2._CTRL16.SIZE:=ANY_TO_WORD(SIZEOF(CTRL2));
CTRL3._CTRL16.SIZE:=ANY_TO_WORD(SIZEOF(CTRL3));
TIMER(IN:=TRUE, PT:=T#500MS);
IF	TIMER.Q THEN
	TIMER(IN:=FALSE);
	CASE STAGE OF
		0:
			SET_BIT16(ADR(CTRL2),N);
			OR16(ADR(CTRL1),ADR(CTRL2),ADR(CTRL3));
			X1 := GET_BIT16(ADR(CTRL1),N);
			X2 := GET_BIT16(ADR(CTRL2),N);
			X3 := GET_BIT16(ADR(CTRL3),N);
			STAGE := 1;
		1:
			RESET_BIT16(ADR(CTRL2),N);
			SET_BIT16(ADR(CTRL1),N);
			OR16(ADR(CTRL1),ADR(CTRL2),ADR(CTRL3));
			X1 := GET_BIT16(ADR(CTRL1),N);
			X2 := GET_BIT16(ADR(CTRL2),N);
			X3 := GET_BIT16(ADR(CTRL3),N);
			STAGE := 2;
		2:
			SET_BIT16(ADR(CTRL2),N);
			OR16(ADR(CTRL1),ADR(CTRL2),ADR(CTRL3));
			X1 := GET_BIT16(ADR(CTRL1),N);
			X2 := GET_BIT16(ADR(CTRL2),N);
			X3 := GET_BIT16(ADR(CTRL3),N);
			STAGE := 3;
		3:
			RESET_BIT16(ADR(CTRL1),N);
			RESET_BIT16(ADR(CTRL2),N);
			OR16(ADR(CTRL1),ADR(CTRL2),ADR(CTRL3));
			X1 := GET_BIT16(ADR(CTRL1),N);
			X2 := GET_BIT16(ADR(CTRL2),N);
			X3 := GET_BIT16(ADR(CTRL3),N);
			STAGE := 0;
			N:=N+1;
			IF	N = 32 THEN
				N := 0;
			END_IF
	END_CASE
END_IF
IF	X3 = (X1 OR X2) THEN
	CORRECT	:=	TRUE;
ELSE
	CORRECT	:=	FALSE;
END_IF
          
END_PROGRAM

PROGRAM CHECK_OR32
  VAR
    CTRL1 : uCTRL32;
    CTRL2 : uCTRL32;
    CTRL3 : uCTRL32;
    TIMER : TON;
    STAGE : ENUM;
    N : LINT;
    X1 : BOOL;
    X2 : BOOL;
    X3 : BOOL;
    CORRECT : BOOL := TRUE;
  END_VAR

            CTRL1._CTRL32.SIZE:=ANY_TO_DWORD(SIZEOF(CTRL1));
CTRL2._CTRL32.SIZE:=ANY_TO_DWORD(SIZEOF(CTRL2));
CTRL3._CTRL32.SIZE:=ANY_TO_DWORD(SIZEOF(CTRL3));
TIMER(IN:=TRUE, PT:=T#500MS);
IF	TIMER.Q THEN
	TIMER(IN:=FALSE);
	CASE STAGE OF
		0:
			SET_BIT32(ADR(CTRL2),N);
			OR32(ADR(CTRL1),ADR(CTRL2),ADR(CTRL3));
			X1 := GET_BIT32(ADR(CTRL1),N);
			X2 := GET_BIT32(ADR(CTRL2),N);
			X3 := GET_BIT32(ADR(CTRL3),N);
			STAGE := 1;
		1:
			RESET_BIT32(ADR(CTRL2),N);
			SET_BIT32(ADR(CTRL1),N);
			OR32(ADR(CTRL1),ADR(CTRL2),ADR(CTRL3));
			X1 := GET_BIT32(ADR(CTRL1),N);
			X2 := GET_BIT32(ADR(CTRL2),N);
			X3 := GET_BIT32(ADR(CTRL3),N);
			STAGE := 2;
		2:
			SET_BIT32(ADR(CTRL2),N);
			OR32(ADR(CTRL1),ADR(CTRL2),ADR(CTRL3));
			X1 := GET_BIT32(ADR(CTRL1),N);
			X2 := GET_BIT32(ADR(CTRL2),N);
			X3 := GET_BIT32(ADR(CTRL3),N);
			STAGE := 3;
		3:
			RESET_BIT32(ADR(CTRL1),N);
			RESET_BIT32(ADR(CTRL2),N);
			OR32(ADR(CTRL1),ADR(CTRL2),ADR(CTRL3));
			X1 := GET_BIT32(ADR(CTRL1),N);
			X2 := GET_BIT32(ADR(CTRL2),N);
			X3 := GET_BIT32(ADR(CTRL3),N);
			STAGE := 0;
			N:=N+1;
			IF	N = 64 THEN
				N := 0;
			END_IF
	END_CASE
END_IF
IF	X3 = (X1 OR X2) THEN
	CORRECT	:=	TRUE;
ELSE
	CORRECT	:=	FALSE;
END_IF
          
END_PROGRAM

PROGRAM CHECK_NEQ32
  VAR
    CTRL1 : uCTRL32;
    CTRL2 : uCTRL32;
    CTRL3 : uCTRL32;
    TIMER : TON;
    STAGE : ENUM;
    N : LINT;
    X1 : BOOL;
    X2 : BOOL;
    X3 : BOOL;
    CORRECT : BOOL := TRUE;
  END_VAR

            CTRL1._CTRL32.SIZE:=ANY_TO_DWORD(SIZEOF(CTRL1));
CTRL2._CTRL32.SIZE:=ANY_TO_DWORD(SIZEOF(CTRL2));
CTRL3._CTRL32.SIZE:=ANY_TO_DWORD(SIZEOF(CTRL3));
TIMER(IN:=TRUE, PT:=T#500MS);
IF	TIMER.Q THEN
	TIMER(IN:=FALSE);
	CASE STAGE OF
		0:
			SET_BIT32(ADR(CTRL2),N);
			NEQ32(ADR(CTRL1),ADR(CTRL2),ADR(CTRL3));
			X1 := GET_BIT32(ADR(CTRL1),N);
			X2 := GET_BIT32(ADR(CTRL2),N);
			X3 := GET_BIT32(ADR(CTRL3),N);
			STAGE := 1;
		1:
			RESET_BIT32(ADR(CTRL2),N);
			SET_BIT32(ADR(CTRL1),N);
			NEQ32(ADR(CTRL1),ADR(CTRL2),ADR(CTRL3));
			X1 := GET_BIT32(ADR(CTRL1),N);
			X2 := GET_BIT32(ADR(CTRL2),N);
			X3 := GET_BIT32(ADR(CTRL3),N);
			STAGE := 2;
		2:
			SET_BIT32(ADR(CTRL2),N);
			NEQ32(ADR(CTRL1),ADR(CTRL2),ADR(CTRL3));
			X1 := GET_BIT32(ADR(CTRL1),N);
			X2 := GET_BIT32(ADR(CTRL2),N);
			X3 := GET_BIT32(ADR(CTRL3),N);
			STAGE := 3;
		3:
			RESET_BIT32(ADR(CTRL1),N);
			RESET_BIT32(ADR(CTRL2),N);
			NEQ32(ADR(CTRL1),ADR(CTRL2),ADR(CTRL3));
			X1 := GET_BIT32(ADR(CTRL1),N);
			X2 := GET_BIT32(ADR(CTRL2),N);
			X3 := GET_BIT32(ADR(CTRL3),N);
			STAGE := 0;
			N:=N+1;
			IF	N = 64 THEN
				N := 0;
			END_IF
	END_CASE
END_IF
IF	X3 = NOT(X1 = X2) THEN
	CORRECT	:=	TRUE;
ELSE
	CORRECT	:=	FALSE;
END_IF
          
END_PROGRAM

FUNCTION FINDNTH_1_32 : LINT
  VAR_INPUT
    IN_ADR1 : POINTER TO WORD;
    N : LINT;
  END_VAR
  VAR
    SIZE : DWORD;
    pdwADR1 : POINTER TO DWORD;
    COUNT : DWORD;
    N_COUNT : LINT := -1;
  END_VAR
  VAR CONSTANT
    ONE : DWORD := 1;
    STEP : DWORD := 4;
    STEP_SIZE : DWORD := (STEP * 8);
  END_VAR

            pdwADR1	:=	IN_ADR1+STEP;
SIZE	:=	pdwADR1^;
FOR COUNT:=2*STEP TO SIZE-1 BY STEP DO
	pdwADR1	:=	IN_ADR1+COUNT;
	IF NOT(pdwADR1^ =0) THEN
		REPEAT
 			IF	(NOT(SHL(ONE,FINDNTH_1_32 MOD STEP_SIZE)) OR pdwADR1^ )= 4294967295 THEN			
				N_COUNT := N_COUNT + 1;
				IF	N_COUNT = N THEN
					RETURN;					
				END_IF 	
			END_IF;
			FINDNTH_1_32:=FINDNTH_1_32 + 1;
		UNTIL FINDNTH_1_32 MOD STEP_SIZE = 0
		END_REPEAT;
	ELSE
		FINDNTH_1_32:=FINDNTH_1_32 + STEP_SIZE;
	END_IF
END_FOR
FINDNTH_1_32:=-1;
          
END_FUNCTION

FUNCTION FINDNTH_0_16 : LINT
  VAR_INPUT
    IN_ADR1 : POINTER TO WORD;
    N : LINT;
  END_VAR
  VAR
    SIZE : WORD;
    pwADR1 : POINTER TO WORD;
    COUNT : WORD;
    N_COUNT : LINT := -1;
  END_VAR
  VAR CONSTANT
    ONE : WORD := 1;
    STEP : WORD := 2;
    STEP_SIZE : WORD := (STEP * 8);
  END_VAR

            pwADR1	:=	IN_ADR1+STEP;
SIZE	:=	pwADR1^;
FOR COUNT:=2*STEP TO SIZE-1 BY STEP DO
	pwADR1	:=	IN_ADR1+COUNT;
		REPEAT
 			IF	NOT((NOT(SHL(ONE,FINDNTH_0_16 MOD STEP_SIZE)) OR pwADR1^ )= 65535) THEN			
				N_COUNT := N_COUNT + 1;
				IF	N_COUNT = N THEN
					RETURN;					
				END_IF 		
			END_IF;
			FINDNTH_0_16:=FINDNTH_0_16 + 1;
		UNTIL FINDNTH_0_16 MOD STEP_SIZE = 0
		END_REPEAT;	
END_FOR
FINDNTH_0_16:=-1;
          
END_FUNCTION

PROGRAM CHECK_NXOR8
  VAR
    CTRL1 : uCTRL8;
    CTRL2 : uCTRL8;
    CTRL3 : uCTRL8;
    TIMER : TON;
    STAGE : ENUM;
    N : LINT;
    X1 : BOOL;
    X2 : BOOL;
    X3 : BOOL;
    CORRECT : BOOL := TRUE;
  END_VAR

            CTRL1._CTRL8.SIZE:=ANY_TO_BYTE(SIZEOF(CTRL1));
CTRL2._CTRL8.SIZE:=ANY_TO_BYTE(SIZEOF(CTRL2));
CTRL3._CTRL8.SIZE:=ANY_TO_BYTE(SIZEOF(CTRL3));
TIMER(IN:=TRUE, PT:=T#500mS);
IF	TIMER.Q THEN
	TIMER(IN:=FALSE);
	CASE STAGE OF
		0:
			SET_BIT8(ADR(CTRL2),N);
			NXOR8(ADR(CTRL1),ADR(CTRL2),ADR(CTRL3));
			X1 := GET_BIT8(ADR(CTRL1),N);
			X2 := GET_BIT8(ADR(CTRL2),N);
			X3 := GET_BIT8(ADR(CTRL3),N);
			STAGE := 1;
		1:
			RESET_BIT8(ADR(CTRL2),N);
			SET_BIT8(ADR(CTRL1),N);
			NXOR8(ADR(CTRL1),ADR(CTRL2),ADR(CTRL3));
			X1 := GET_BIT8(ADR(CTRL1),N);
			X2 := GET_BIT8(ADR(CTRL2),N);
			X3 := GET_BIT8(ADR(CTRL3),N);
			STAGE := 2;
		2:
			SET_BIT8(ADR(CTRL2),N);
			NXOR8(ADR(CTRL1),ADR(CTRL2),ADR(CTRL3));
			X1 := GET_BIT8(ADR(CTRL1),N);
			X2 := GET_BIT8(ADR(CTRL2),N);
			X3 := GET_BIT8(ADR(CTRL3),N);
			STAGE := 3;
		3:
			RESET_BIT8(ADR(CTRL1),N);
			RESET_BIT8(ADR(CTRL2),N);
			NXOR8(ADR(CTRL1),ADR(CTRL2),ADR(CTRL3));
			X1 := GET_BIT8(ADR(CTRL1),N);
			X2 := GET_BIT8(ADR(CTRL2),N);
			X3 := GET_BIT8(ADR(CTRL3),N);
			STAGE := 0;
			N:=N+1;
			IF	N = 16 THEN
				N := 0;
			END_IF
	END_CASE
END_IF
IF	X3 = NOT (X1 XOR X2) THEN
	CORRECT	:=	TRUE;
ELSE
	CORRECT	:=	FALSE;
END_IF
          
END_PROGRAM

PROGRAM CHECK_NXOR16
  VAR
    CTRL1 : uCTRL16;
    CTRL2 : uCTRL16;
    CTRL3 : uCTRL16;
    TIMER : TON;
    STAGE : ENUM;
    N : LINT;
    X1 : BOOL;
    X2 : BOOL;
    X3 : BOOL;
    CORRECT : BOOL := TRUE;
  END_VAR

            CTRL1._CTRL16.SIZE:=ANY_TO_WORD(SIZEOF(CTRL1));
CTRL2._CTRL16.SIZE:=ANY_TO_WORD(SIZEOF(CTRL2));
CTRL3._CTRL16.SIZE:=ANY_TO_WORD(SIZEOF(CTRL3));
TIMER(IN:=TRUE, PT:=T#500MS);
IF	TIMER.Q THEN
	TIMER(IN:=FALSE);
	CASE STAGE OF
		0:
			SET_BIT16(ADR(CTRL2),N);
			NXOR16(ADR(CTRL1),ADR(CTRL2),ADR(CTRL3));
			X1 := GET_BIT16(ADR(CTRL1),N);
			X2 := GET_BIT16(ADR(CTRL2),N);
			X3 := GET_BIT16(ADR(CTRL3),N);
			STAGE := 1;
		1:
			RESET_BIT16(ADR(CTRL2),N);
			SET_BIT16(ADR(CTRL1),N);
			NXOR16(ADR(CTRL1),ADR(CTRL2),ADR(CTRL3));
			X1 := GET_BIT16(ADR(CTRL1),N);
			X2 := GET_BIT16(ADR(CTRL2),N);
			X3 := GET_BIT16(ADR(CTRL3),N);
			STAGE := 2;
		2:
			SET_BIT16(ADR(CTRL2),N);
			NXOR16(ADR(CTRL1),ADR(CTRL2),ADR(CTRL3));
			X1 := GET_BIT16(ADR(CTRL1),N);
			X2 := GET_BIT16(ADR(CTRL2),N);
			X3 := GET_BIT16(ADR(CTRL3),N);
			STAGE := 3;
		3:
			RESET_BIT16(ADR(CTRL1),N);
			RESET_BIT16(ADR(CTRL2),N);
			NXOR16(ADR(CTRL1),ADR(CTRL2),ADR(CTRL3));
			X1 := GET_BIT16(ADR(CTRL1),N);
			X2 := GET_BIT16(ADR(CTRL2),N);
			X3 := GET_BIT16(ADR(CTRL3),N);
			STAGE := 0;
			N:=N+1;
			IF	N = 32 THEN
				N := 0;
			END_IF
	END_CASE
END_IF
IF	X3 = NOT (X1 XOR X2) THEN
	CORRECT	:=	TRUE;
ELSE
	CORRECT	:=	FALSE;
END_IF
          
END_PROGRAM

PROGRAM CHECK_NXOR32
  VAR
    CTRL1 : uCTRL32;
    CTRL2 : uCTRL32;
    CTRL3 : uCTRL32;
    TIMER : TON;
    STAGE : ENUM;
    N : LINT;
    X1 : BOOL;
    X2 : BOOL;
    X3 : BOOL;
    CORRECT : BOOL := TRUE;
  END_VAR

            CTRL1._CTRL32.SIZE:=ANY_TO_DWORD(SIZEOF(CTRL1));
CTRL2._CTRL32.SIZE:=ANY_TO_DWORD(SIZEOF(CTRL2));
CTRL3._CTRL32.SIZE:=ANY_TO_DWORD(SIZEOF(CTRL3));
TIMER(IN:=TRUE, PT:=T#500MS);
IF	TIMER.Q THEN
	TIMER(IN:=FALSE);
	CASE STAGE OF
		0:
			SET_BIT32(ADR(CTRL2),N);
			NXOR32(ADR(CTRL1),ADR(CTRL2),ADR(CTRL3));
			X1 := GET_BIT32(ADR(CTRL1),N);
			X2 := GET_BIT32(ADR(CTRL2),N);
			X3 := GET_BIT32(ADR(CTRL3),N);
			STAGE := 1;
		1:
			RESET_BIT32(ADR(CTRL2),N);
			SET_BIT32(ADR(CTRL1),N);
			NXOR32(ADR(CTRL1),ADR(CTRL2),ADR(CTRL3));
			X1 := GET_BIT32(ADR(CTRL1),N);
			X2 := GET_BIT32(ADR(CTRL2),N);
			X3 := GET_BIT32(ADR(CTRL3),N);
			STAGE := 2;
		2:
			SET_BIT32(ADR(CTRL2),N);
			NXOR32(ADR(CTRL1),ADR(CTRL2),ADR(CTRL3));
			X1 := GET_BIT32(ADR(CTRL1),N);
			X2 := GET_BIT32(ADR(CTRL2),N);
			X3 := GET_BIT32(ADR(CTRL3),N);
			STAGE := 3;
		3:
			RESET_BIT32(ADR(CTRL1),N);
			RESET_BIT32(ADR(CTRL2),N);
			NXOR32(ADR(CTRL1),ADR(CTRL2),ADR(CTRL3));
			X1 := GET_BIT32(ADR(CTRL1),N);
			X2 := GET_BIT32(ADR(CTRL2),N);
			X3 := GET_BIT32(ADR(CTRL3),N);
			STAGE := 0;
			N:=N+1;
			IF	N = 64 THEN
				N := 0;
			END_IF
	END_CASE
END_IF
IF	X3 = NOT (X1 XOR X2) THEN
	CORRECT	:=	TRUE;
ELSE
	CORRECT	:=	FALSE;
END_IF
          
END_PROGRAM

PROGRAM CHECK_NOR8
  VAR
    CTRL1 : uCTRL8;
    CTRL2 : uCTRL8;
    CTRL3 : uCTRL8;
    TIMER : TON;
    STAGE : ENUM;
    N : LINT;
    X1 : BOOL;
    X2 : BOOL;
    X3 : BOOL;
    CORRECT : BOOL := TRUE;
  END_VAR

            CTRL1._CTRL8.SIZE:=ANY_TO_BYTE(SIZEOF(CTRL1));
CTRL2._CTRL8.SIZE:=ANY_TO_BYTE(SIZEOF(CTRL2));
CTRL3._CTRL8.SIZE:=ANY_TO_BYTE(SIZEOF(CTRL3));
TIMER(IN:=TRUE, PT:=T#500mS);
IF	TIMER.Q THEN
	TIMER(IN:=FALSE);
	CASE STAGE OF
		0:
			SET_BIT8(ADR(CTRL2),N);
			NOR8(ADR(CTRL1),ADR(CTRL2),ADR(CTRL3));
			X1 := GET_BIT8(ADR(CTRL1),N);
			X2 := GET_BIT8(ADR(CTRL2),N);
			X3 := GET_BIT8(ADR(CTRL3),N);
			STAGE := 1;
		1:
			RESET_BIT8(ADR(CTRL2),N);
			SET_BIT8(ADR(CTRL1),N);
			NOR8(ADR(CTRL1),ADR(CTRL2),ADR(CTRL3));
			X1 := GET_BIT8(ADR(CTRL1),N);
			X2 := GET_BIT8(ADR(CTRL2),N);
			X3 := GET_BIT8(ADR(CTRL3),N);
			STAGE := 2;
		2:
			SET_BIT8(ADR(CTRL2),N);
			NOR8(ADR(CTRL1),ADR(CTRL2),ADR(CTRL3));
			X1 := GET_BIT8(ADR(CTRL1),N);
			X2 := GET_BIT8(ADR(CTRL2),N);
			X3 := GET_BIT8(ADR(CTRL3),N);
			STAGE := 3;
		3:
			RESET_BIT8(ADR(CTRL1),N);
			RESET_BIT8(ADR(CTRL2),N);
			NOR8(ADR(CTRL1),ADR(CTRL2),ADR(CTRL3));
			X1 := GET_BIT8(ADR(CTRL1),N);
			X2 := GET_BIT8(ADR(CTRL2),N);
			X3 := GET_BIT8(ADR(CTRL3),N);
			STAGE := 0;
			N:=N+1;
			IF	N = 16 THEN
				N := 0;
			END_IF
	END_CASE
END_IF
IF	X3 = NOT(X1 OR X2) THEN
	CORRECT	:=	TRUE;
ELSE
	CORRECT	:=	FALSE;
END_IF
          
END_PROGRAM

PROGRAM CHECK_NOR16
  VAR
    CTRL1 : uCTRL16;
    CTRL2 : uCTRL16;
    CTRL3 : uCTRL16;
    TIMER : TON;
    STAGE : ENUM;
    N : LINT;
    X1 : BOOL;
    X2 : BOOL;
    X3 : BOOL;
    CORRECT : BOOL := TRUE;
  END_VAR

            CTRL1._CTRL16.SIZE:=ANY_TO_WORD(SIZEOF(CTRL1));
CTRL2._CTRL16.SIZE:=ANY_TO_WORD(SIZEOF(CTRL2));
CTRL3._CTRL16.SIZE:=ANY_TO_WORD(SIZEOF(CTRL3));
TIMER(IN:=TRUE, PT:=T#500MS);
IF	TIMER.Q THEN
	TIMER(IN:=FALSE);
	CASE STAGE OF
		0:
			SET_BIT16(ADR(CTRL2),N);
			NOR16(ADR(CTRL1),ADR(CTRL2),ADR(CTRL3));
			X1 := GET_BIT16(ADR(CTRL1),N);
			X2 := GET_BIT16(ADR(CTRL2),N);
			X3 := GET_BIT16(ADR(CTRL3),N);
			STAGE := 1;
		1:
			RESET_BIT16(ADR(CTRL2),N);
			SET_BIT16(ADR(CTRL1),N);
			NOR16(ADR(CTRL1),ADR(CTRL2),ADR(CTRL3));
			X1 := GET_BIT16(ADR(CTRL1),N);
			X2 := GET_BIT16(ADR(CTRL2),N);
			X3 := GET_BIT16(ADR(CTRL3),N);
			STAGE := 2;
		2:
			SET_BIT16(ADR(CTRL2),N);
			NOR16(ADR(CTRL1),ADR(CTRL2),ADR(CTRL3));
			X1 := GET_BIT16(ADR(CTRL1),N);
			X2 := GET_BIT16(ADR(CTRL2),N);
			X3 := GET_BIT16(ADR(CTRL3),N);
			STAGE := 3;
		3:
			RESET_BIT16(ADR(CTRL1),N);
			RESET_BIT16(ADR(CTRL2),N);
			NOR16(ADR(CTRL1),ADR(CTRL2),ADR(CTRL3));
			X1 := GET_BIT16(ADR(CTRL1),N);
			X2 := GET_BIT16(ADR(CTRL2),N);
			X3 := GET_BIT16(ADR(CTRL3),N);
			STAGE := 0;
			N:=N+1;
			IF	N = 32 THEN
				N := 0;
			END_IF
	END_CASE
END_IF
IF	X3 = NOT(X1 OR X2) THEN
	CORRECT	:=	TRUE;
ELSE
	CORRECT	:=	FALSE;
END_IF
          
END_PROGRAM

PROGRAM CHECK_NOR32
  VAR
    CTRL1 : uCTRL32;
    CTRL2 : uCTRL32;
    CTRL3 : uCTRL32;
    TIMER : TON;
    STAGE : ENUM;
    N : LINT;
    X1 : BOOL;
    X2 : BOOL;
    X3 : BOOL;
    CORRECT : BOOL := TRUE;
  END_VAR

            CTRL1._CTRL32.SIZE:=ANY_TO_DWORD(SIZEOF(CTRL1));
CTRL2._CTRL32.SIZE:=ANY_TO_DWORD(SIZEOF(CTRL2));
CTRL3._CTRL32.SIZE:=ANY_TO_DWORD(SIZEOF(CTRL3));
TIMER(IN:=TRUE, PT:=T#500MS);
IF	TIMER.Q THEN
	TIMER(IN:=FALSE);
	CASE STAGE OF
		0:
			SET_BIT32(ADR(CTRL2),N);
			NOR32(ADR(CTRL1),ADR(CTRL2),ADR(CTRL3));
			X1 := GET_BIT32(ADR(CTRL1),N);
			X2 := GET_BIT32(ADR(CTRL2),N);
			X3 := GET_BIT32(ADR(CTRL3),N);
			STAGE := 1;
		1:
			RESET_BIT32(ADR(CTRL2),N);
			SET_BIT32(ADR(CTRL1),N);
			NOR32(ADR(CTRL1),ADR(CTRL2),ADR(CTRL3));
			X1 := GET_BIT32(ADR(CTRL1),N);
			X2 := GET_BIT32(ADR(CTRL2),N);
			X3 := GET_BIT32(ADR(CTRL3),N);
			STAGE := 2;
		2:
			SET_BIT32(ADR(CTRL2),N);
			NOR32(ADR(CTRL1),ADR(CTRL2),ADR(CTRL3));
			X1 := GET_BIT32(ADR(CTRL1),N);
			X2 := GET_BIT32(ADR(CTRL2),N);
			X3 := GET_BIT32(ADR(CTRL3),N);
			STAGE := 3;
		3:
			RESET_BIT32(ADR(CTRL1),N);
			RESET_BIT32(ADR(CTRL2),N);
			NOR32(ADR(CTRL1),ADR(CTRL2),ADR(CTRL3));
			X1 := GET_BIT32(ADR(CTRL1),N);
			X2 := GET_BIT32(ADR(CTRL2),N);
			X3 := GET_BIT32(ADR(CTRL3),N);
			STAGE := 0;
			N:=N+1;
			IF	N = 64 THEN
				N := 0;
			END_IF
	END_CASE
END_IF
IF	X3 = NOT(X1 OR X2) THEN
	CORRECT	:=	TRUE;
ELSE
	CORRECT	:=	FALSE;
END_IF
          
END_PROGRAM

FUNCTION FINDNTH_0_32 : LINT
  VAR_INPUT
    IN_ADR1 : POINTER TO DWORD;
    N : LINT;
  END_VAR
  VAR
    SIZE : DWORD;
    pdwADR1 : POINTER TO DWORD;
    COUNT : DWORD;
    N_COUNT : LINT := -1;
  END_VAR
  VAR CONSTANT
    ONE : DWORD := 1;
    STEP : DWORD := 4;
    STEP_SIZE : DWORD := (STEP * 8);
  END_VAR

            pdwADR1	:=	IN_ADR1+STEP;
SIZE	:=	pdwADR1^;
FOR COUNT:=2*STEP TO SIZE-1 BY STEP DO
	pdwADR1	:=	IN_ADR1+COUNT;
		REPEAT
 			IF	NOT((NOT(SHL(ONE,FINDNTH_0_32 MOD STEP_SIZE)) OR pdwADR1^ )= 4294967295) THEN		
				N_COUNT := N_COUNT + 1;
				IF	N_COUNT = N THEN
					RETURN;					
				END_IF 			
			END_IF;
			FINDNTH_0_32:=FINDNTH_0_32 + 1;
		UNTIL FINDNTH_0_32 MOD STEP_SIZE = 0
		END_REPEAT;	
END_FOR
FINDNTH_0_32:=-1;
          
END_FUNCTION

PROGRAM CHECK_XOR8
  VAR
    CTRL1 : uCTRL8;
    CTRL2 : uCTRL8;
    CTRL3 : uCTRL8;
    TIMER : TON;
    STAGE : ENUM;
    N : LINT;
    X1 : BOOL;
    X2 : BOOL;
    X3 : BOOL;
    CORRECT : BOOL := TRUE;
  END_VAR

            CTRL1._CTRL8.SIZE:=ANY_TO_BYTE(SIZEOF(CTRL1));
CTRL2._CTRL8.SIZE:=ANY_TO_BYTE(SIZEOF(CTRL2));
CTRL3._CTRL8.SIZE:=ANY_TO_BYTE(SIZEOF(CTRL3));
TIMER(IN:=TRUE, PT:=T#500mS);
IF	TIMER.Q THEN
	TIMER(IN:=FALSE);
	CASE STAGE OF
		0:
			SET_BIT8(ADR(CTRL2),N);
			XOR8(ADR(CTRL1),ADR(CTRL2),ADR(CTRL3));
			X1 := GET_BIT8(ADR(CTRL1),N);
			X2 := GET_BIT8(ADR(CTRL2),N);
			X3 := GET_BIT8(ADR(CTRL3),N);
			STAGE := 1;
		1:
			RESET_BIT8(ADR(CTRL2),N);
			SET_BIT8(ADR(CTRL1),N);
			XOR8(ADR(CTRL1),ADR(CTRL2),ADR(CTRL3));
			X1 := GET_BIT8(ADR(CTRL1),N);
			X2 := GET_BIT8(ADR(CTRL2),N);
			X3 := GET_BIT8(ADR(CTRL3),N);
			STAGE := 2;
		2:
			SET_BIT8(ADR(CTRL2),N);
			XOR8(ADR(CTRL1),ADR(CTRL2),ADR(CTRL3));
			X1 := GET_BIT8(ADR(CTRL1),N);
			X2 := GET_BIT8(ADR(CTRL2),N);
			X3 := GET_BIT8(ADR(CTRL3),N);
			STAGE := 3;
		3:
			RESET_BIT8(ADR(CTRL1),N);
			RESET_BIT8(ADR(CTRL2),N);
			XOR8(ADR(CTRL1),ADR(CTRL2),ADR(CTRL3));
			X1 := GET_BIT8(ADR(CTRL1),N);
			X2 := GET_BIT8(ADR(CTRL2),N);
			X3 := GET_BIT8(ADR(CTRL3),N);
			STAGE := 0;
			N:=N+1;
			IF	N = 16 THEN
				N := 0;
			END_IF
	END_CASE
END_IF
IF	X3 = (X1 XOR X2) THEN
	CORRECT	:=	TRUE;
ELSE
	CORRECT	:=	FALSE;
END_IF
          
END_PROGRAM

PROGRAM CHECK_XOR16
  VAR
    CTRL1 : uCTRL16;
    CTRL2 : uCTRL16;
    CTRL3 : uCTRL16;
    TIMER : TON;
    STAGE : ENUM;
    N : LINT;
    X1 : BOOL;
    X2 : BOOL;
    X3 : BOOL;
    CORRECT : BOOL := TRUE;
  END_VAR

            CTRL1._CTRL16.SIZE:=ANY_TO_WORD(SIZEOF(CTRL1));
CTRL2._CTRL16.SIZE:=ANY_TO_WORD(SIZEOF(CTRL2));
CTRL3._CTRL16.SIZE:=ANY_TO_WORD(SIZEOF(CTRL3));
TIMER(IN:=TRUE, PT:=T#500MS);
IF	TIMER.Q THEN
	TIMER(IN:=FALSE);
	CASE STAGE OF
		0:
			SET_BIT16(ADR(CTRL2),N);
			XOR16(ADR(CTRL1),ADR(CTRL2),ADR(CTRL3));
			X1 := GET_BIT16(ADR(CTRL1),N);
			X2 := GET_BIT16(ADR(CTRL2),N);
			X3 := GET_BIT16(ADR(CTRL3),N);
			STAGE := 1;
		1:
			RESET_BIT16(ADR(CTRL2),N);
			SET_BIT16(ADR(CTRL1),N);
			XOR16(ADR(CTRL1),ADR(CTRL2),ADR(CTRL3));
			X1 := GET_BIT16(ADR(CTRL1),N);
			X2 := GET_BIT16(ADR(CTRL2),N);
			X3 := GET_BIT16(ADR(CTRL3),N);
			STAGE := 2;
		2:
			SET_BIT16(ADR(CTRL2),N);
			XOR16(ADR(CTRL1),ADR(CTRL2),ADR(CTRL3));
			X1 := GET_BIT16(ADR(CTRL1),N);
			X2 := GET_BIT16(ADR(CTRL2),N);
			X3 := GET_BIT16(ADR(CTRL3),N);
			STAGE := 3;
		3:
			RESET_BIT16(ADR(CTRL1),N);
			RESET_BIT16(ADR(CTRL2),N);
			XOR16(ADR(CTRL1),ADR(CTRL2),ADR(CTRL3));
			X1 := GET_BIT16(ADR(CTRL1),N);
			X2 := GET_BIT16(ADR(CTRL2),N);
			X3 := GET_BIT16(ADR(CTRL3),N);
			STAGE := 0;
			N:=N+1;
			IF	N = 32 THEN
				N := 0;
			END_IF
	END_CASE
END_IF
IF	X3 = (X1 XOR X2) THEN
	CORRECT	:=	TRUE;
ELSE
	CORRECT	:=	FALSE;
END_IF
          
END_PROGRAM

PROGRAM CHECK_XOR32
  VAR
    CTRL1 : uCTRL32;
    CTRL2 : uCTRL32;
    CTRL3 : uCTRL32;
    TIMER : TON;
    STAGE : ENUM;
    N : LINT;
    X1 : BOOL;
    X2 : BOOL;
    X3 : BOOL;
    CORRECT : BOOL := TRUE;
  END_VAR

            CTRL1._CTRL32.SIZE:=ANY_TO_DWORD(SIZEOF(CTRL1));
CTRL2._CTRL32.SIZE:=ANY_TO_DWORD(SIZEOF(CTRL2));
CTRL3._CTRL32.SIZE:=ANY_TO_DWORD(SIZEOF(CTRL3));
TIMER(IN:=TRUE, PT:=T#500MS);
IF	TIMER.Q THEN
	TIMER(IN:=FALSE);
	CASE STAGE OF
		0:
			SET_BIT32(ADR(CTRL2),N);
			XOR32(ADR(CTRL1),ADR(CTRL2),ADR(CTRL3));
			X1 := GET_BIT32(ADR(CTRL1),N);
			X2 := GET_BIT32(ADR(CTRL2),N);
			X3 := GET_BIT32(ADR(CTRL3),N);
			STAGE := 1;
		1:
			RESET_BIT32(ADR(CTRL2),N);
			SET_BIT32(ADR(CTRL1),N);
			XOR32(ADR(CTRL1),ADR(CTRL2),ADR(CTRL3));
			X1 := GET_BIT32(ADR(CTRL1),N);
			X2 := GET_BIT32(ADR(CTRL2),N);
			X3 := GET_BIT32(ADR(CTRL3),N);
			STAGE := 2;
		2:
			SET_BIT32(ADR(CTRL2),N);
			XOR32(ADR(CTRL1),ADR(CTRL2),ADR(CTRL3));
			X1 := GET_BIT32(ADR(CTRL1),N);
			X2 := GET_BIT32(ADR(CTRL2),N);
			X3 := GET_BIT32(ADR(CTRL3),N);
			STAGE := 3;
		3:
			RESET_BIT32(ADR(CTRL1),N);
			RESET_BIT32(ADR(CTRL2),N);
			XOR32(ADR(CTRL1),ADR(CTRL2),ADR(CTRL3));
			X1 := GET_BIT32(ADR(CTRL1),N);
			X2 := GET_BIT32(ADR(CTRL2),N);
			X3 := GET_BIT32(ADR(CTRL3),N);
			STAGE := 0;
			N:=N+1;
			IF	N = 64 THEN
				N := 0;
			END_IF
	END_CASE
END_IF
IF	X3 = (X1 XOR X2) THEN
	CORRECT	:=	TRUE;
ELSE
	CORRECT	:=	FALSE;
END_IF
          
END_PROGRAM

PROGRAM CHECK_NOT8
  VAR
    CTRL1 : uCTRL8;
    CTRL2 : uCTRL8;
    TIMER : TON;
    STAGE : ENUM;
    N : LINT;
    X1 : BOOL;
    X2 : BOOL;
    CORRECT : BOOL := TRUE;
  END_VAR

            CTRL1._CTRL8.SIZE:=ANY_TO_BYTE(SIZEOF(CTRL1));
CTRL2._CTRL8.SIZE:=ANY_TO_BYTE(SIZEOF(CTRL2));
TIMER(IN:=TRUE, PT:=T#500MS);
IF	TIMER.Q THEN
	TIMER(IN:=FALSE);
	CASE STAGE OF
		0:
			SET_BIT8(ADR(CTRL1),N);
			NOT8(ADR(CTRL1),ADR(CTRL2));
			X1 := GET_BIT8(ADR(CTRL1),N);
			X2 := GET_BIT8(ADR(CTRL2),N);
			STAGE := 1;
		1:
			RESET_BIT8(ADR(CTRL1),N);
			NOT8(ADR(CTRL1),ADR(CTRL2));
			X1 := GET_BIT8(ADR(CTRL1),N);
			X2 := GET_BIT8(ADR(CTRL2),N);
			STAGE := 0;
			N:=N+1;
			IF	N = 16 THEN
				N := 0;
			END_IF
	END_CASE
END_IF
IF	X2 = NOT X1 THEN
	CORRECT	:=	TRUE;
ELSE
	CORRECT	:=	FALSE;
END_IF
          
END_PROGRAM

PROGRAM CHECK_NOT16
  VAR
    CTRL1 : uCTRL16;
    CTRL2 : uCTRL16;
    TIMER : TON;
    STAGE : ENUM;
    N : LINT;
    X1 : BOOL;
    X2 : BOOL;
    CORRECT : BOOL := TRUE;
  END_VAR

            CTRL1._CTRL16.SIZE:=ANY_TO_WORD(SIZEOF(CTRL1));
CTRL2._CTRL16.SIZE:=ANY_TO_WORD(SIZEOF(CTRL2));
TIMER(IN:=TRUE, PT:=T#500MS);
IF	TIMER.Q THEN
	TIMER(IN:=FALSE);
	CASE STAGE OF
		0:
			SET_BIT16(ADR(CTRL1),N);
			NOT16(ADR(CTRL1),ADR(CTRL2));
			X1 := GET_BIT16(ADR(CTRL1),N);
			X2 := GET_BIT16(ADR(CTRL2),N);
			STAGE := 1;
		1:
			RESET_BIT16(ADR(CTRL1),N);
			NOT16(ADR(CTRL1),ADR(CTRL2));
			X1 := GET_BIT16(ADR(CTRL1),N);
			X2 := GET_BIT16(ADR(CTRL2),N);
			STAGE := 0;
			N:=N+1;
			IF	N = 32 THEN
				N := 0;
			END_IF
	END_CASE
END_IF
IF	X2 = NOT X1 THEN
	CORRECT	:=	TRUE;
ELSE
	CORRECT	:=	FALSE;
END_IF
          
END_PROGRAM

PROGRAM CHECK_NOT32
  VAR
    CTRL1 : uCTRL32;
    CTRL2 : uCTRL32;
    TIMER : TON;
    STAGE : ENUM;
    N : LINT;
    X1 : BOOL;
    X2 : BOOL;
    CORRECT : BOOL := TRUE;
  END_VAR

            CTRL1._CTRL32.SIZE:=ANY_TO_DWORD(SIZEOF(CTRL1));
CTRL2._CTRL32.SIZE:=ANY_TO_DWORD(SIZEOF(CTRL2));
TIMER(IN:=TRUE, PT:=T#500MS);
IF	TIMER.Q THEN
	TIMER(IN:=FALSE);
	CASE STAGE OF
		0:
			SET_BIT32(ADR(CTRL1),N);
			NOT32(ADR(CTRL1),ADR(CTRL2));
			X1 := GET_BIT32(ADR(CTRL1),N);
			X2 := GET_BIT32(ADR(CTRL2),N);
			STAGE := 1;
		1:
			RESET_BIT32(ADR(CTRL1),N);
			NOT32(ADR(CTRL1),ADR(CTRL2));
			X1 := GET_BIT32(ADR(CTRL1),N);
			X2 := GET_BIT32(ADR(CTRL2),N);
			STAGE := 0;
			N:=N+1;
			IF	N = 64 THEN
				N := 0;
			END_IF
	END_CASE
END_IF
IF	X2 = NOT X1 THEN
	CORRECT	:=	TRUE;
ELSE
	CORRECT	:=	FALSE;
END_IF
          
END_PROGRAM

FUNCTION FINDNTH_0_8 : LINT
  VAR_INPUT
    IN_ADR1 : POINTER TO BYTE;
    N : LINT;
  END_VAR
  VAR
    SIZE : BYTE;
    pbADR1 : POINTER TO BYTE;
    COUNT : BYTE;
    N_COUNT : LINT := -1;
  END_VAR
  VAR CONSTANT
    ONE : BYTE := 1;
  END_VAR

            pbADR1	:=	IN_ADR1+1;
SIZE	:=	pbADR1^;
FOR COUNT:=2 TO SIZE-1 DO
	pbADR1	:=	IN_ADR1+COUNT;
		REPEAT
 			IF	NOT((NOT(SHL(ONE,FINDNTH_0_8 MOD 8)) OR pbADR1^ )= 255) THEN
				N_COUNT := N_COUNT + 1;
				IF	N_COUNT = N THEN
					RETURN;					
				END_IF
			END_IF;
			FINDNTH_0_8:=FINDNTH_0_8 + 1;
		UNTIL FINDNTH_0_8 MOD 8 = 0
		END_REPEAT;	
END_FOR
FINDNTH_0_8:=-1;
          
END_FUNCTION

PROGRAM CHECK_FINDNTH_0_8
  VAR
    CTRL1 : uCTRL8;
    N : LINT;
    M : LINT;
  END_VAR

            CTRL1._CTRL8.SIZE:=ANY_TO_BYTE(SIZEOF(CTRL1));
M:=FINDNTH_0_8(ADR(CTRL1),N);
          
END_PROGRAM

PROGRAM CHECK_FINDNTH_0_16
  VAR
    CTRL1 : uCTRL16;
    N : LINT;
    M : LINT;
  END_VAR

            CTRL1._CTRL16.SIZE:=ANY_TO_BYTE(SIZEOF(CTRL1));
M:=FINDNTH_0_16(ADR(CTRL1),N);
          
END_PROGRAM

PROGRAM CHECK_FINDNTH_0_32
  VAR
    CTRL1 : uCTRL32;
    N : LINT;
    M : LINT;
  END_VAR

            CTRL1._CTRL32.SIZE:=ANY_TO_BYTE(SIZEOF(CTRL1));
M:=FINDNTH_0_32(ADR(CTRL1),N);
          
END_PROGRAM

FUNCTION FINDNTH_1_8 : LINT
  VAR_INPUT
    IN_ADR1 : POINTER TO BYTE;
    N : LINT;
  END_VAR
  VAR
    SIZE : BYTE;
    pbADR1 : POINTER TO BYTE;
    COUNT : BYTE;
    N_COUNT : LINT := -1;
  END_VAR
  VAR CONSTANT
    ONE : BYTE := 1;
    STEP : BYTE := 1;
    STEP_SIZE : BYTE := (STEP * 8);
  END_VAR

            pbADR1	:=	IN_ADR1+STEP;
SIZE	:=	pbADR1^;
FOR COUNT:=2 TO SIZE-1 DO
	pbADR1	:=	IN_ADR1+COUNT;
	IF NOT(pbADR1^ =0) THEN
		REPEAT
 			IF	(NOT(SHL(ONE,FINDNTH_1_8 MOD 8)) OR pbADR1^ )= 255 THEN			
				N_COUNT := N_COUNT + 1;
				IF	N_COUNT = N THEN
					RETURN;					
				END_IF 	
			END_IF;
			FINDNTH_1_8:=FINDNTH_1_8 + 1;
		UNTIL FINDNTH_1_8 MOD 8 = 0
		END_REPEAT;
	ELSE
		FINDNTH_1_8:=FINDNTH_1_8 + 8;
	END_IF
END_FOR
FINDNTH_1_8:=-1;
          
END_FUNCTION

PROGRAM CHECK_FINDNTH_1_8
  VAR
    CTRL1 : uCTRL8;
    N : LINT;
    M : LINT;
  END_VAR

            CTRL1._CTRL8.SIZE:=ANY_TO_BYTE(SIZEOF(CTRL1));
M:=FINDNTH_1_8(ADR(CTRL1),N);
          
END_PROGRAM

FUNCTION FINDNTH_1_16 : LINT
  VAR_INPUT
    IN_ADR1 : POINTER TO WORD;
    N : LINT;
  END_VAR
  VAR
    SIZE : WORD;
    pwADR1 : POINTER TO WORD;
    COUNT : WORD;
    N_COUNT : LINT := -1;
  END_VAR
  VAR CONSTANT
    ONE : WORD := 1;
    STEP : WORD := 2;
    STEP_SIZE : WORD := (STEP * 8);
  END_VAR

            pwADR1	:=	IN_ADR1+STEP;
SIZE	:=	pwADR1^;
FOR COUNT:=2*STEP TO SIZE-STEP BY STEP DO
	pwADR1	:=	IN_ADR1+COUNT;
	IF NOT(pwADR1^ =0) THEN
		REPEAT
 			IF	(NOT(SHL(ONE,FINDNTH_1_16 MOD STEP_SIZE)) OR pwADR1^ )= 65535 THEN 			
				N_COUNT := N_COUNT + 1;
				IF	N_COUNT = N THEN
					RETURN;					
				END_IF 	
			END_IF;
			FINDNTH_1_16:=FINDNTH_1_16 + 1;
		UNTIL FINDNTH_1_16 MOD STEP_SIZE = 0
		END_REPEAT;
	ELSE
		FINDNTH_1_16:=FINDNTH_1_16 + STEP_SIZE;
	END_IF
END_FOR
FINDNTH_1_16:=-1;
          
END_FUNCTION

PROGRAM CHECK_FINDNTH_1_16
  VAR
    CTRL1 : uCTRL16;
    N : LINT;
    M : LINT;
  END_VAR

            CTRL1._CTRL16.SIZE:=ANY_TO_BYTE(SIZEOF(CTRL1));
M:=FINDNTH_1_16(ADR(CTRL1),N);
          
END_PROGRAM

PROGRAM CHECK_FINDNTH_1_32
  VAR
    CTRL1 : uCTRL32;
    N : LINT;
    M : LINT;
  END_VAR

            CTRL1._CTRL32.SIZE:=ANY_TO_BYTE(SIZEOF(CTRL1));
M:=FINDNTH_1_32(ADR(CTRL1),N);
          
END_PROGRAM
